      movel([0.344723, -1.349574, -2.579464, -0.783351, 1.570796, 1.915519],accel_mss,speed_ms,0,blend_radius_m)
      speed_ms = 0.003
      movel([0.344723, -1.359446, -2.584078, -0.768865, 1.570796, 1.915519],accel_mss,speed_ms,0,blend_radius_m)
      speed_ms = 0.007
      movel([0.344029, -1.359514, -2.584032, -0.768843, 1.570796, 1.914825],accel_mss,speed_ms,0,blend_radius_m)
      movel([0.343242, -1.359584, -2.583985, -0.768820, 1.570796, 1.914038],accel_mss,speed_ms,0,blend_radius_m)
      movel([0.342310, -1.359660, -2.583934, -0.768796, 1.570796, 1.913106],accel_mss,speed_ms,0,blend_radius_m)
      movel([0.339886, -1.359848, -2.583806, -0.768735, 1.570796, 1.910682],accel_mss,speed_ms,0,blend_radius_m)
      movel([0.340151, -1.359124, -2.584296, -0.768969, 1.570796, 1.910947],accel_mss,speed_ms,0,blend_radius_m)
      movel([0.340416, -1.358401, -2.584784, -0.769203, 1.570796, 1.911212],accel_mss,speed_ms,0,blend_radius_m)
      movel([0.342598, -1.358879, -2.584462, -0.769048, 1.570796, 1.913394],accel_mss,speed_ms,0,blend_radius_m)
      movel([0.343434, -1.359066, -2.584335, -0.768988, 1.570796, 1.914230],accel_mss,speed_ms,0,blend_radius_m)
      movel([0.344132, -1.359235, -2.584221, -0.768933, 1.570796, 1.914929],accel_mss,speed_ms,0,blend_radius_m)
      movel([0.344743, -1.359392, -2.584115, -0.768882, 1.570796, 1.915539],accel_mss,speed_ms,0,blend_radius_m)
      movel([0.344756, -1.359400, -2.584109, -0.768880, 1.570796, 1.915553],accel_mss,speed_ms,0,blend_radius_m)
      movel([0.344754, -1.359419, -2.584097, -0.768874, 1.570796, 1.915551],accel_mss,speed_ms,0,blend_radius_m)
      movel([0.344743, -1.359435, -2.584085, -0.768868, 1.570796, 1.915540],accel_mss,speed_ms,0,blend_radius_m)
      movel([0.344723, -1.359446, -2.584078, -0.768865, 1.570796, 1.915519],accel_mss,speed_ms,0,blend_radius_m)
      speed_ms = 0.003
      movel([0.344723, -1.362784, -2.585600, -0.764005, 1.570796, 1.915519],accel_mss,speed_ms,0,blend_radius_m)
      speed_ms = 0.007
      movel([0.344029, -1.362852, -2.585554, -0.763984, 1.570796, 1.914825],accel_mss,speed_ms,0,blend_radius_m)
      movel([0.343242, -1.362922, -2.585506, -0.763961, 1.570796, 1.914038],accel_mss,speed_ms,0,blend_radius_m)
      movel([0.342310, -1.362997, -2.585455, -0.763937, 1.570796, 1.913106],accel_mss,speed_ms,0,blend_radius_m)
      movel([0.339886, -1.363185, -2.585327, -0.763877, 1.570796, 1.910682],accel_mss,speed_ms,0,blend_radius_m)
      movel([0.340151, -1.362463, -2.585818, -0.764108, 1.570796, 1.910947],accel_mss,speed_ms,0,blend_radius_m)
      movel([0.340416, -1.361742, -2.586307, -0.764340, 1.570796, 1.911212],accel_mss,speed_ms,0,blend_radius_m)
      movel([0.342598, -1.362219, -2.585984, -0.764186, 1.570796, 1.913394],accel_mss,speed_ms,0,blend_radius_m)
      movel([0.343434, -1.362405, -2.585857, -0.764127, 1.570796, 1.914230],accel_mss,speed_ms,0,blend_radius_m)
      movel([0.344132, -1.362573, -2.585743, -0.764073, 1.570796, 1.914929],accel_mss,speed_ms,0,blend_radius_m)
      movel([0.344743, -1.362730, -2.585636, -0.764022, 1.570796, 1.915539],accel_mss,speed_ms,0,blend_radius_m)
      movel([0.344756, -1.362738, -2.585631, -0.764020, 1.570796, 1.915553],accel_mss,speed_ms,0,blend_radius_m)
      movel([0.344754, -1.362757, -2.585618, -0.764014, 1.570796, 1.915551],accel_mss,speed_ms,0,blend_radius_m)
      movel([0.344743, -1.362773, -2.585607, -0.764009, 1.570796, 1.915540],accel_mss,speed_ms,0,blend_radius_m)
      movel([0.344723, -1.362784, -2.585600, -0.764005, 1.570796, 1.915519],accel_mss,speed_ms,0,blend_radius_m)
      speed_ms = 0.003
      movel([0.344723, -1.349574, -2.579464, -0.783351, 1.570796, 1.915519],accel_mss,speed_ms,0,blend_radius_m)
      speed_ms = 0.01
      movel([0.344723, -1.324283, -2.566799, -0.821307, 1.570796, 1.915519],accel_mss,speed_ms,0,blend_radius_m)
      movel([0.344980, -1.321488, -2.568590, -0.822311, 1.570796, 1.915776],accel_mss,speed_ms,0,blend_radius_m)
      movel([0.344980, -1.346826, -2.581290, -0.784273, 1.570796, 1.915776],accel_mss,speed_ms,0,blend_radius_m)
      speed_ms = 0.003
      movel([0.344980, -1.356718, -2.585918, -0.769752, 1.570796, 1.915776],accel_mss,speed_ms,0,blend_radius_m)
      speed_ms = 0.007
      movel([0.344880, -1.356721, -2.585916, -0.769751, 1.570796, 1.915676],accel_mss,speed_ms,0,blend_radius_m)
      movel([0.344783, -1.356715, -2.585921, -0.769754, 1.570796, 1.915579],accel_mss,speed_ms,0,blend_radius_m)
      movel([0.344690, -1.356699, -2.585931, -0.769759, 1.570796, 1.915486],accel_mss,speed_ms,0,blend_radius_m)
      movel([0.320621, -1.351621, -2.589329, -0.771439, 1.570796, 1.891418],accel_mss,speed_ms,0,blend_radius_m)
      movel([0.295950, -1.347201, -2.592258, -0.772930, 1.570796, 1.866746],accel_mss,speed_ms,0,blend_radius_m)
      movel([0.295898, -1.347189, -2.592266, -0.772934, 1.570796, 1.866695],accel_mss,speed_ms,0,blend_radius_m)
      movel([0.295858, -1.347164, -2.592282, -0.772943, 1.570796, 1.866654],accel_mss,speed_ms,0,blend_radius_m)
      movel([0.295822, -1.347135, -2.592301, -0.772953, 1.570796, 1.866618],accel_mss,speed_ms,0,blend_radius_m)
      movel([0.295809, -1.347107, -2.592320, -0.772962, 1.570796, 1.866606],accel_mss,speed_ms,0,blend_radius_m)
      movel([0.295812, -1.347070, -2.592344, -0.772975, 1.570796, 1.866608],accel_mss,speed_ms,0,blend_radius_m)
      movel([0.295826, -1.347031, -2.592369, -0.772988, 1.570796, 1.866623],accel_mss,speed_ms,0,blend_radius_m)
      movel([0.300073, -1.339721, -2.597152, -0.775516, 1.570796, 1.870870],accel_mss,speed_ms,0,blend_radius_m)
      movel([0.304360, -1.332369, -2.601889, -0.778132, 1.570796, 1.875156],accel_mss,speed_ms,0,blend_radius_m)
      movel([0.304408, -1.332297, -2.601935, -0.778157, 1.570796, 1.875204],accel_mss,speed_ms,0,blend_radius_m)
      movel([0.304466, -1.332229, -2.601978, -0.778182, 1.570796, 1.875263],accel_mss,speed_ms,0,blend_radius_m)
      movel([0.304533, -1.332167, -2.602018, -0.778204, 1.570796, 1.875329],accel_mss,speed_ms,0,blend_radius_m)
      movel([0.304566, -1.332146, -2.602031, -0.778212, 1.570796, 1.875363],accel_mss,speed_ms,0,blend_radius_m)
      movel([0.304602, -1.332142, -2.602034, -0.778213, 1.570796, 1.875398],accel_mss,speed_ms,0,blend_radius_m)
      movel([0.306078, -1.332291, -2.601938, -0.778159, 1.570796, 1.876875],accel_mss,speed_ms,0,blend_radius_m)
      movel([0.307729, -1.332470, -2.601824, -0.778095, 1.570796, 1.878525],accel_mss,speed_ms,0,blend_radius_m)
      movel([0.309667, -1.332702, -2.601676, -0.778011, 1.570796, 1.880463],accel_mss,speed_ms,0,blend_radius_m)
      movel([0.315690, -1.333471, -2.601183, -0.777735, 1.570796, 1.886487],accel_mss,speed_ms,0,blend_radius_m)
      movel([0.321678, -1.334295, -2.600655, -0.777439, 1.570796, 1.892474],accel_mss,speed_ms,0,blend_radius_m)
      movel([0.323791, -1.334609, -2.600453, -0.777327, 1.570796, 1.894587],accel_mss,speed_ms,0,blend_radius_m)
      movel([0.325891, -1.334945, -2.600237, -0.777207, 1.570796, 1.896687],accel_mss,speed_ms,0,blend_radius_m)
      movel([0.327973, -1.335306, -2.600005, -0.777078, 1.570796, 1.898769],accel_mss,speed_ms,0,blend_radius_m)
      movel([0.329039, -1.335506, -2.599877, -0.777006, 1.570796, 1.899836],accel_mss,speed_ms,0,blend_radius_m)
      movel([0.330096, -1.335717, -2.599741, -0.776931, 1.570796, 1.900893],accel_mss,speed_ms,0,blend_radius_m)
      movel([0.331144, -1.335944, -2.599595, -0.776850, 1.570796, 1.901941],accel_mss,speed_ms,0,blend_radius_m)
      movel([0.332182, -1.336185, -2.599439, -0.776764, 1.570796, 1.902978],accel_mss,speed_ms,0,blend_radius_m)
      movel([0.333127, -1.336420, -2.599288, -0.776681, 1.570796, 1.903923],accel_mss,speed_ms,0,blend_radius_m)
      movel([0.334059, -1.336671, -2.599126, -0.776592, 1.570796, 1.904855],accel_mss,speed_ms,0,blend_radius_m)
      movel([0.334978, -1.336941, -2.598952, -0.776496, 1.570796, 1.905774],accel_mss,speed_ms,0,blend_radius_m)
      movel([0.335887, -1.337224, -2.598769, -0.776396, 1.570796, 1.906684],accel_mss,speed_ms,0,blend_radius_m)
      movel([0.336686, -1.337490, -2.598597, -0.776302, 1.570796, 1.907483],accel_mss,speed_ms,0,blend_radius_m)
      movel([0.337471, -1.337775, -2.598413, -0.776201, 1.570796, 1.908267],accel_mss,speed_ms,0,blend_radius_m)
      movel([0.338245, -1.338072, -2.598221, -0.776096, 1.570796, 1.909041],accel_mss,speed_ms,0,blend_radius_m)
      movel([0.339005, -1.338388, -2.598016, -0.775984, 1.570796, 1.909801],accel_mss,speed_ms,0,blend_radius_m)
      movel([0.339755, -1.338718, -2.597803, -0.775868, 1.570796, 1.910551],accel_mss,speed_ms,0,blend_radius_m)
      movel([0.340490, -1.339065, -2.597578, -0.775746, 1.570796, 1.911286],accel_mss,speed_ms,0,blend_radius_m)
      movel([0.341213, -1.339426, -2.597344, -0.775619, 1.570796, 1.912009],accel_mss,speed_ms,0,blend_radius_m)
      movel([0.341919, -1.339803, -2.597099, -0.775487, 1.570796, 1.912715],accel_mss,speed_ms,0,blend_radius_m)
      movel([0.342412, -1.340083, -2.596917, -0.775389, 1.570796, 1.913209],accel_mss,speed_ms,0,blend_radius_m)
      movel([0.342888, -1.340385, -2.596721, -0.775283, 1.570796, 1.913685],accel_mss,speed_ms,0,blend_radius_m)
      movel([0.343349, -1.340701, -2.596515, -0.775173, 1.570796, 1.914145],accel_mss,speed_ms,0,blend_radius_m)
      movel([0.343790, -1.341036, -2.596297, -0.775056, 1.570796, 1.914586],accel_mss,speed_ms,0,blend_radius_m)
      movel([0.344215, -1.341389, -2.596067, -0.774933, 1.570796, 1.915011],accel_mss,speed_ms,0,blend_radius_m)
      movel([0.344625, -1.341755, -2.595829, -0.774805, 1.570796, 1.915421],accel_mss,speed_ms,0,blend_radius_m)
      movel([0.345013, -1.342139, -2.595579, -0.774672, 1.570796, 1.915809],accel_mss,speed_ms,0,blend_radius_m)
      movel([0.345385, -1.342540, -2.595316, -0.774532, 1.570796, 1.916181],accel_mss,speed_ms,0,blend_radius_m)
      movel([0.345737, -1.342955, -2.595045, -0.774388, 1.570796, 1.916534],accel_mss,speed_ms,0,blend_radius_m)
      movel([0.345992, -1.343283, -2.594831, -0.774275, 1.570796, 1.916789],accel_mss,speed_ms,0,blend_radius_m)
      movel([0.346229, -1.343625, -2.594607, -0.774157, 1.570796, 1.917026],accel_mss,speed_ms,0,blend_radius_m)
      movel([0.346450, -1.343978, -2.594376, -0.774035, 1.570796, 1.917247],accel_mss,speed_ms,0,blend_radius_m)
      movel([0.346655, -1.344344, -2.594136, -0.773909, 1.570796, 1.917451],accel_mss,speed_ms,0,blend_radius_m)
      movel([0.346843, -1.344721, -2.593889, -0.773779, 1.570796, 1.917639],accel_mss,speed_ms,0,blend_radius_m)
      movel([0.347014, -1.345108, -2.593635, -0.773646, 1.570796, 1.917811],accel_mss,speed_ms,0,blend_radius_m)
      movel([0.347168, -1.345505, -2.593374, -0.773510, 1.570796, 1.917964],accel_mss,speed_ms,0,blend_radius_m)
      movel([0.347305, -1.345913, -2.593106, -0.773370, 1.570796, 1.918102],accel_mss,speed_ms,0,blend_radius_m)
      movel([0.347424, -1.346332, -2.592830, -0.773227, 1.570796, 1.918221],accel_mss,speed_ms,0,blend_radius_m)
      movel([0.347525, -1.346761, -2.592548, -0.773080, 1.570796, 1.918321],accel_mss,speed_ms,0,blend_radius_m)
      movel([0.347605, -1.347180, -2.592272, -0.772938, 1.570796, 1.918401],accel_mss,speed_ms,0,blend_radius_m)
      movel([0.347668, -1.347607, -2.591990, -0.772792, 1.570796, 1.918464],accel_mss,speed_ms,0,blend_radius_m)
      movel([0.347707, -1.348044, -2.591701, -0.772644, 1.570796, 1.918504],accel_mss,speed_ms,0,blend_radius_m)
      movel([0.347731, -1.348488, -2.591408, -0.772493, 1.570796, 1.918527],accel_mss,speed_ms,0,blend_radius_m)
      movel([0.347733, -1.348942, -2.591108, -0.772340, 1.570796, 1.918529],accel_mss,speed_ms,0,blend_radius_m)
      movel([0.347720, -1.349399, -2.590805, -0.772185, 1.570796, 1.918516],accel_mss,speed_ms,0,blend_radius_m)
      movel([0.347684, -1.349864, -2.590496, -0.772028, 1.570796, 1.918481],accel_mss,speed_ms,0,blend_radius_m)
      movel([0.347630, -1.350336, -2.590184, -0.771870, 1.570796, 1.918426],accel_mss,speed_ms,0,blend_radius_m)
      movel([0.347558, -1.350810, -2.589868, -0.771710, 1.570796, 1.918354],accel_mss,speed_ms,0,blend_radius_m)
      movel([0.347467, -1.351290, -2.589549, -0.771549, 1.570796, 1.918263],accel_mss,speed_ms,0,blend_radius_m)
      movel([0.347400, -1.351565, -2.589366, -0.771457, 1.570796, 1.918196],accel_mss,speed_ms,0,blend_radius_m)
      movel([0.347318, -1.351842, -2.589182, -0.771365, 1.570796, 1.918115],accel_mss,speed_ms,0,blend_radius_m)
      movel([0.347219, -1.352121, -2.588996, -0.771272, 1.570796, 1.918015],accel_mss,speed_ms,0,blend_radius_m)
      movel([0.346861, -1.353037, -2.588385, -0.770967, 1.570796, 1.917658],accel_mss,speed_ms,0,blend_radius_m)
      movel([0.346494, -1.353953, -2.587773, -0.770663, 1.570796, 1.917291],accel_mss,speed_ms,0,blend_radius_m)
      movel([0.346110, -1.354891, -2.587145, -0.770353, 1.570796, 1.916906],accel_mss,speed_ms,0,blend_radius_m)
      movel([0.345719, -1.355829, -2.586516, -0.770044, 1.570796, 1.916515],accel_mss,speed_ms,0,blend_radius_m)
      movel([0.345654, -1.355967, -2.586424, -0.769999, 1.570796, 1.916450],accel_mss,speed_ms,0,blend_radius_m)
      movel([0.345581, -1.356105, -2.586331, -0.769953, 1.570796, 1.916377],accel_mss,speed_ms,0,blend_radius_m)
      movel([0.345495, -1.356240, -2.586240, -0.769909, 1.570796, 1.916292],accel_mss,speed_ms,0,blend_radius_m)
      movel([0.345403, -1.356375, -2.586149, -0.769865, 1.570796, 1.916199],accel_mss,speed_ms,0,blend_radius_m)
      movel([0.345351, -1.356438, -2.586107, -0.769844, 1.570796, 1.916147],accel_mss,speed_ms,0,blend_radius_m)
      movel([0.345294, -1.356502, -2.586064, -0.769823, 1.570796, 1.916090],accel_mss,speed_ms,0,blend_radius_m)
      movel([0.345238, -1.356559, -2.586025, -0.769804, 1.570796, 1.916034],accel_mss,speed_ms,0,blend_radius_m)
      movel([0.345175, -1.356612, -2.585990, -0.769787, 1.570796, 1.915972],accel_mss,speed_ms,0,blend_radius_m)
      movel([0.345123, -1.356652, -2.585963, -0.769774, 1.570796, 1.915919],accel_mss,speed_ms,0,blend_radius_m)
      movel([0.345067, -1.356689, -2.585938, -0.769762, 1.570796, 1.915863],accel_mss,speed_ms,0,blend_radius_m)
      movel([0.345023, -1.356710, -2.585924, -0.769755, 1.570796, 1.915820],accel_mss,speed_ms,0,blend_radius_m)
      movel([0.344980, -1.356718, -2.585918, -0.769752, 1.570796, 1.915776],accel_mss,speed_ms,0,blend_radius_m)
      speed_ms = 0.003
      movel([0.344980, -1.360063, -2.587444, -0.764881, 1.570796, 1.915776],accel_mss,speed_ms,0,blend_radius_m)
      speed_ms = 0.007
      movel([0.344880, -1.360066, -2.587442, -0.764880, 1.570796, 1.915676],accel_mss,speed_ms,0,blend_radius_m)
      movel([0.344783, -1.360060, -2.587447, -0.764882, 1.570796, 1.915579],accel_mss,speed_ms,0,blend_radius_m)
      movel([0.344690, -1.360044, -2.587457, -0.764888, 1.570796, 1.915486],accel_mss,speed_ms,0,blend_radius_m)
      movel([0.320621, -1.354979, -2.590864, -0.766546, 1.570796, 1.891418],accel_mss,speed_ms,0,blend_radius_m)
      movel([0.295950, -1.350570, -2.593800, -0.768019, 1.570796, 1.866746],accel_mss,speed_ms,0,blend_radius_m)
      movel([0.295898, -1.350559, -2.593807, -0.768023, 1.570796, 1.866695],accel_mss,speed_ms,0,blend_radius_m)
      movel([0.295858, -1.350534, -2.593824, -0.768031, 1.570796, 1.866654],accel_mss,speed_ms,0,blend_radius_m)
      movel([0.295822, -1.350504, -2.593843, -0.768041, 1.570796, 1.866618],accel_mss,speed_ms,0,blend_radius_m)
      movel([0.295809, -1.350476, -2.593862, -0.768051, 1.570796, 1.866606],accel_mss,speed_ms,0,blend_radius_m)
      movel([0.295812, -1.350440, -2.593886, -0.768063, 1.570796, 1.866608],accel_mss,speed_ms,0,blend_radius_m)
      movel([0.295826, -1.350401, -2.593912, -0.768076, 1.570796, 1.866623],accel_mss,speed_ms,0,blend_radius_m)
      movel([0.300073, -1.343109, -2.598706, -0.770573, 1.570796, 1.870870],accel_mss,speed_ms,0,blend_radius_m)
      movel([0.304360, -1.335775, -2.603456, -0.773158, 1.570796, 1.875156],accel_mss,speed_ms,0,blend_radius_m)
      movel([0.304408, -1.335704, -2.603501, -0.773184, 1.570796, 1.875204],accel_mss,speed_ms,0,blend_radius_m)
      movel([0.304466, -1.335636, -2.603545, -0.773208, 1.570796, 1.875263],accel_mss,speed_ms,0,blend_radius_m)
      movel([0.304533, -1.335574, -2.603585, -0.773230, 1.570796, 1.875329],accel_mss,speed_ms,0,blend_radius_m)
      movel([0.304566, -1.335553, -2.603598, -0.773238, 1.570796, 1.875363],accel_mss,speed_ms,0,blend_radius_m)
      movel([0.304602, -1.335549, -2.603601, -0.773239, 1.570796, 1.875398],accel_mss,speed_ms,0,blend_radius_m)
      movel([0.306078, -1.335698, -2.603505, -0.773186, 1.570796, 1.876875],accel_mss,speed_ms,0,blend_radius_m)
      movel([0.307729, -1.335876, -2.603390, -0.773122, 1.570796, 1.878525],accel_mss,speed_ms,0,blend_radius_m)
      movel([0.309667, -1.336108, -2.603242, -0.773040, 1.570796, 1.880463],accel_mss,speed_ms,0,blend_radius_m)
      movel([0.315690, -1.336875, -2.602748, -0.772766, 1.570796, 1.886487],accel_mss,speed_ms,0,blend_radius_m)
      movel([0.321678, -1.337697, -2.602218, -0.772474, 1.570796, 1.892474],accel_mss,speed_ms,0,blend_radius_m)
      movel([0.323791, -1.338010, -2.602016, -0.772363, 1.570796, 1.894587],accel_mss,speed_ms,0,blend_radius_m)
      movel([0.325891, -1.338345, -2.601800, -0.772244, 1.570796, 1.896687],accel_mss,speed_ms,0,blend_radius_m)
      movel([0.327973, -1.338705, -2.601567, -0.772117, 1.570796, 1.898769],accel_mss,speed_ms,0,blend_radius_m)
      movel([0.329039, -1.338904, -2.601438, -0.772046, 1.570796, 1.899836],accel_mss,speed_ms,0,blend_radius_m)
      movel([0.330096, -1.339115, -2.601302, -0.771972, 1.570796, 1.900893],accel_mss,speed_ms,0,blend_radius_m)
      movel([0.331144, -1.339342, -2.601155, -0.771892, 1.570796, 1.901941],accel_mss,speed_ms,0,blend_radius_m)
      movel([0.332182, -1.339582, -2.600999, -0.771807, 1.570796, 1.902978],accel_mss,speed_ms,0,blend_radius_m)
      movel([0.333127, -1.339817, -2.600848, -0.771725, 1.570796, 1.903923],accel_mss,speed_ms,0,blend_radius_m)
      movel([0.334059, -1.340067, -2.600685, -0.771637, 1.570796, 1.904855],accel_mss,speed_ms,0,blend_radius_m)
      movel([0.334978, -1.340336, -2.600511, -0.771542, 1.570796, 1.905774],accel_mss,speed_ms,0,blend_radius_m)
      movel([0.335887, -1.340619, -2.600328, -0.771443, 1.570796, 1.906684],accel_mss,speed_ms,0,blend_radius_m)
      movel([0.336686, -1.340884, -2.600155, -0.771350, 1.570796, 1.907483],accel_mss,speed_ms,0,blend_radius_m)
      movel([0.337471, -1.341168, -2.599971, -0.771250, 1.570796, 1.908267],accel_mss,speed_ms,0,blend_radius_m)
      movel([0.338245, -1.341465, -2.599778, -0.771146, 1.570796, 1.909041],accel_mss,speed_ms,0,blend_radius_m)
      movel([0.339005, -1.341780, -2.599573, -0.771036, 1.570796, 1.909801],accel_mss,speed_ms,0,blend_radius_m)
      movel([0.339755, -1.342108, -2.599359, -0.770922, 1.570796, 1.910551],accel_mss,speed_ms,0,blend_radius_m)
      movel([0.340490, -1.342455, -2.599133, -0.770801, 1.570796, 1.911286],accel_mss,speed_ms,0,blend_radius_m)
      movel([0.341213, -1.342815, -2.598899, -0.770676, 1.570796, 1.912009],accel_mss,speed_ms,0,blend_radius_m)
      movel([0.341919, -1.343191, -2.598653, -0.770545, 1.570796, 1.912715],accel_mss,speed_ms,0,blend_radius_m)
      movel([0.342412, -1.343471, -2.598471, -0.770448, 1.570796, 1.913209],accel_mss,speed_ms,0,blend_radius_m)
      movel([0.342888, -1.343771, -2.598274, -0.770343, 1.570796, 1.913685],accel_mss,speed_ms,0,blend_radius_m)
      movel([0.343349, -1.344087, -2.598068, -0.770234, 1.570796, 1.914145],accel_mss,speed_ms,0,blend_radius_m)
      movel([0.343790, -1.344421, -2.597849, -0.770118, 1.570796, 1.914586],accel_mss,speed_ms,0,blend_radius_m)
      movel([0.344215, -1.344773, -2.597619, -0.769997, 1.570796, 1.915011],accel_mss,speed_ms,0,blend_radius_m)
      movel([0.344625, -1.345138, -2.597380, -0.769871, 1.570796, 1.915421],accel_mss,speed_ms,0,blend_radius_m)
      movel([0.345013, -1.345521, -2.597129, -0.769739, 1.570796, 1.915809],accel_mss,speed_ms,0,blend_radius_m)
      movel([0.345385, -1.345922, -2.596866, -0.769601, 1.570796, 1.916181],accel_mss,speed_ms,0,blend_radius_m)
      movel([0.345737, -1.346336, -2.596594, -0.769459, 1.570796, 1.916534],accel_mss,speed_ms,0,blend_radius_m)
      movel([0.345992, -1.346662, -2.596380, -0.769347, 1.570796, 1.916789],accel_mss,speed_ms,0,blend_radius_m)
      movel([0.346229, -1.347004, -2.596155, -0.769230, 1.570796, 1.917026],accel_mss,speed_ms,0,blend_radius_m)
      movel([0.346450, -1.347356, -2.595923, -0.769110, 1.570796, 1.917247],accel_mss,speed_ms,0,blend_radius_m)
      movel([0.346655, -1.347721, -2.595683, -0.768985, 1.570796, 1.917451],accel_mss,speed_ms,0,blend_radius_m)
      movel([0.346843, -1.348097, -2.595435, -0.768857, 1.570796, 1.917639],accel_mss,speed_ms,0,blend_radius_m)
      movel([0.347014, -1.348483, -2.595180, -0.768726, 1.570796, 1.917811],accel_mss,speed_ms,0,blend_radius_m)
      movel([0.347168, -1.348879, -2.594919, -0.768591, 1.570796, 1.917964],accel_mss,speed_ms,0,blend_radius_m)
      movel([0.347305, -1.349286, -2.594650, -0.768453, 1.570796, 1.918102],accel_mss,speed_ms,0,blend_radius_m)
      movel([0.347424, -1.349704, -2.594374, -0.768312, 1.570796, 1.918221],accel_mss,speed_ms,0,blend_radius_m)
      movel([0.347525, -1.350132, -2.594090, -0.768167, 1.570796, 1.918321],accel_mss,speed_ms,0,blend_radius_m)
      movel([0.347605, -1.350549, -2.593813, -0.768026, 1.570796, 1.918401],accel_mss,speed_ms,0,blend_radius_m)
      movel([0.347668, -1.350975, -2.593531, -0.767883, 1.570796, 1.918464],accel_mss,speed_ms,0,blend_radius_m)
      movel([0.347707, -1.351412, -2.593241, -0.767736, 1.570796, 1.918504],accel_mss,speed_ms,0,blend_radius_m)
      movel([0.347731, -1.351854, -2.592948, -0.767587, 1.570796, 1.918527],accel_mss,speed_ms,0,blend_radius_m)
      movel([0.347733, -1.352307, -2.592646, -0.767436, 1.570796, 1.918529],accel_mss,speed_ms,0,blend_radius_m)
      movel([0.347720, -1.352763, -2.592343, -0.767283, 1.570796, 1.918516],accel_mss,speed_ms,0,blend_radius_m)
      movel([0.347684, -1.353227, -2.592034, -0.767128, 1.570796, 1.918481],accel_mss,speed_ms,0,blend_radius_m)
      movel([0.347630, -1.353697, -2.591720, -0.766972, 1.570796, 1.918426],accel_mss,speed_ms,0,blend_radius_m)
      movel([0.347558, -1.354170, -2.591404, -0.766814, 1.570796, 1.918354],accel_mss,speed_ms,0,blend_radius_m)
      movel([0.347467, -1.354649, -2.591084, -0.766655, 1.570796, 1.918263],accel_mss,speed_ms,0,blend_radius_m)
      movel([0.347400, -1.354924, -2.590901, -0.766564, 1.570796, 1.918196],accel_mss,speed_ms,0,blend_radius_m)
      movel([0.347318, -1.355199, -2.590716, -0.766473, 1.570796, 1.918115],accel_mss,speed_ms,0,blend_radius_m)
      movel([0.347219, -1.355478, -2.590530, -0.766381, 1.570796, 1.918015],accel_mss,speed_ms,0,blend_radius_m)
      movel([0.346861, -1.356392, -2.589917, -0.766080, 1.570796, 1.917658],accel_mss,speed_ms,0,blend_radius_m)
      movel([0.346494, -1.357305, -2.589304, -0.765780, 1.570796, 1.917291],accel_mss,speed_ms,0,blend_radius_m)
      movel([0.346110, -1.358241, -2.588674, -0.765474, 1.570796, 1.916906],accel_mss,speed_ms,0,blend_radius_m)
      movel([0.345719, -1.359176, -2.588044, -0.765169, 1.570796, 1.916515],accel_mss,speed_ms,0,blend_radius_m)
      movel([0.345654, -1.359314, -2.587951, -0.765124, 1.570796, 1.916450],accel_mss,speed_ms,0,blend_radius_m)
      movel([0.345581, -1.359452, -2.587858, -0.765080, 1.570796, 1.916377],accel_mss,speed_ms,0,blend_radius_m)
      movel([0.345495, -1.359586, -2.587767, -0.765036, 1.570796, 1.916292],accel_mss,speed_ms,0,blend_radius_m)
      movel([0.345403, -1.359721, -2.587676, -0.764992, 1.570796, 1.916199],accel_mss,speed_ms,0,blend_radius_m)
      movel([0.345351, -1.359784, -2.587633, -0.764972, 1.570796, 1.916147],accel_mss,speed_ms,0,blend_radius_m)
      movel([0.345294, -1.359848, -2.587590, -0.764951, 1.570796, 1.916090],accel_mss,speed_ms,0,blend_radius_m)
      movel([0.345238, -1.359905, -2.587552, -0.764933, 1.570796, 1.916034],accel_mss,speed_ms,0,blend_radius_m)
      movel([0.345175, -1.359957, -2.587516, -0.764916, 1.570796, 1.915972],accel_mss,speed_ms,0,blend_radius_m)
      movel([0.345123, -1.359998, -2.587489, -0.764903, 1.570796, 1.915919],accel_mss,speed_ms,0,blend_radius_m)
      movel([0.345067, -1.360034, -2.587464, -0.764891, 1.570796, 1.915863],accel_mss,speed_ms,0,blend_radius_m)
      movel([0.345023, -1.360055, -2.587450, -0.764884, 1.570796, 1.915820],accel_mss,speed_ms,0,blend_radius_m)
      movel([0.344980, -1.360063, -2.587444, -0.764881, 1.570796, 1.915776],accel_mss,speed_ms,0,blend_radius_m)
      speed_ms = 0.003
      movel([0.344980, -1.346826, -2.581290, -0.784273, 1.570796, 1.915776],accel_mss,speed_ms,0,blend_radius_m)
      speed_ms = 0.01
      movel([0.344980, -1.321488, -2.568590, -0.822311, 1.570796, 1.915776],accel_mss,speed_ms,0,blend_radius_m)
      movel([0.342353, -1.326735, -2.565220, -0.820435, 1.570796, 1.913150],accel_mss,speed_ms,0,blend_radius_m)
      movel([0.342353, -1.351985, -2.577853, -0.782552, 1.570796, 1.913150],accel_mss,speed_ms,0,blend_radius_m)
      speed_ms = 0.003
      movel([0.342353, -1.361839, -2.582456, -0.768095, 1.570796, 1.913150],accel_mss,speed_ms,0,blend_radius_m)
      speed_ms = 0.007
      movel([0.341641, -1.363771, -2.581139, -0.767479, 1.570796, 1.912437],accel_mss,speed_ms,0,blend_radius_m)
      movel([0.340931, -1.365698, -2.579822, -0.766870, 1.570796, 1.911728],accel_mss,speed_ms,0,blend_radius_m)
      movel([0.336123, -1.366174, -2.579495, -0.766720, 1.570796, 1.906919],accel_mss,speed_ms,0,blend_radius_m)
      movel([0.334430, -1.366357, -2.579369, -0.766663, 1.570796, 1.905226],accel_mss,speed_ms,0,blend_radius_m)
      movel([0.332727, -1.366563, -2.579228, -0.766598, 1.570796, 1.903523],accel_mss,speed_ms,0,blend_radius_m)
      movel([0.331393, -1.366752, -2.579098, -0.766539, 1.570796, 1.902189],accel_mss,speed_ms,0,blend_radius_m)
      movel([0.330047, -1.366975, -2.578945, -0.766469, 1.570796, 1.900843],accel_mss,speed_ms,0,blend_radius_m)
      movel([0.328764, -1.367221, -2.578776, -0.766392, 1.570796, 1.899560],accel_mss,speed_ms,0,blend_radius_m)
      movel([0.327473, -1.367502, -2.578582, -0.766304, 1.570796, 1.898270],accel_mss,speed_ms,0,blend_radius_m)
      movel([0.325956, -1.367865, -2.578333, -0.766191, 1.570796, 1.896752],accel_mss,speed_ms,0,blend_radius_m)
      movel([0.324433, -1.368257, -2.578063, -0.766069, 1.570796, 1.895230],accel_mss,speed_ms,0,blend_radius_m)
      movel([0.323162, -1.368604, -2.577824, -0.765961, 1.570796, 1.893958],accel_mss,speed_ms,0,blend_radius_m)
      movel([0.321888, -1.368978, -2.577566, -0.765845, 1.570796, 1.892684],accel_mss,speed_ms,0,blend_radius_m)
      movel([0.320612, -1.369374, -2.577293, -0.765722, 1.570796, 1.891408],accel_mss,speed_ms,0,blend_radius_m)
      movel([0.319335, -1.369795, -2.577002, -0.765592, 1.570796, 1.890132],accel_mss,speed_ms,0,blend_radius_m)
      movel([0.318059, -1.370240, -2.576694, -0.765455, 1.570796, 1.888855],accel_mss,speed_ms,0,blend_radius_m)
      movel([0.316792, -1.370704, -2.576373, -0.765312, 1.570796, 1.887588],accel_mss,speed_ms,0,blend_radius_m)
      movel([0.315526, -1.371191, -2.576035, -0.765162, 1.570796, 1.886322],accel_mss,speed_ms,0,blend_radius_m)
      movel([0.314261, -1.371704, -2.575680, -0.765005, 1.570796, 1.885058],accel_mss,speed_ms,0,blend_radius_m)
      movel([0.312998, -1.372237, -2.575310, -0.764842, 1.570796, 1.883794],accel_mss,speed_ms,0,blend_radius_m)
      movel([0.311739, -1.372792, -2.574924, -0.764673, 1.570796, 1.882536],accel_mss,speed_ms,0,blend_radius_m)
      movel([0.310506, -1.373361, -2.574529, -0.764500, 1.570796, 1.881302],accel_mss,speed_ms,0,blend_radius_m)
      movel([0.309278, -1.373949, -2.574119, -0.764321, 1.570796, 1.880074],accel_mss,speed_ms,0,blend_radius_m)
      movel([0.308056, -1.374560, -2.573693, -0.764136, 1.570796, 1.878852],accel_mss,speed_ms,0,blend_radius_m)
      movel([0.306839, -1.375192, -2.573251, -0.763945, 1.570796, 1.877635],accel_mss,speed_ms,0,blend_radius_m)
      movel([0.305626, -1.375845, -2.572795, -0.763749, 1.570796, 1.876423],accel_mss,speed_ms,0,blend_radius_m)
      movel([0.304459, -1.376497, -2.572338, -0.763554, 1.570796, 1.875255],accel_mss,speed_ms,0,blend_radius_m)
      movel([0.303297, -1.377173, -2.571865, -0.763352, 1.570796, 1.874093],accel_mss,speed_ms,0,blend_radius_m)
      movel([0.302144, -1.377865, -2.571378, -0.763145, 1.570796, 1.872941],accel_mss,speed_ms,0,blend_radius_m)
      movel([0.301002, -1.378581, -2.570875, -0.762933, 1.570796, 1.871798],accel_mss,speed_ms,0,blend_radius_m)
      movel([0.299869, -1.379313, -2.570360, -0.762716, 1.570796, 1.870665],accel_mss,speed_ms,0,blend_radius_m)
      movel([0.299135, -1.379808, -2.570010, -0.762570, 1.570796, 1.869931],accel_mss,speed_ms,0,blend_radius_m)
      movel([0.298406, -1.380316, -2.569652, -0.762421, 1.570796, 1.869202],accel_mss,speed_ms,0,blend_radius_m)
      movel([0.297686, -1.380836, -2.569285, -0.762268, 1.570796, 1.868482],accel_mss,speed_ms,0,blend_radius_m)
      movel([0.296342, -1.381838, -2.568576, -0.761975, 1.570796, 1.867138],accel_mss,speed_ms,0,blend_radius_m)
      movel([0.295013, -1.382858, -2.567853, -0.761678, 1.570796, 1.865810],accel_mss,speed_ms,0,blend_radius_m)
      movel([0.293697, -1.383898, -2.567114, -0.761377, 1.570796, 1.864493],accel_mss,speed_ms,0,blend_radius_m)
      movel([0.292396, -1.384952, -2.566363, -0.761074, 1.570796, 1.863193],accel_mss,speed_ms,0,blend_radius_m)
      movel([0.291708, -1.385525, -2.565955, -0.760909, 1.570796, 1.862504],accel_mss,speed_ms,0,blend_radius_m)
      movel([0.291033, -1.386110, -2.565537, -0.760742, 1.570796, 1.861829],accel_mss,speed_ms,0,blend_radius_m)
      movel([0.290369, -1.386703, -2.565113, -0.760573, 1.570796, 1.861165],accel_mss,speed_ms,0,blend_radius_m)
      movel([0.289528, -1.387480, -2.564557, -0.760352, 1.570796, 1.860324],accel_mss,speed_ms,0,blend_radius_m)
      movel([0.288705, -1.388267, -2.563993, -0.760129, 1.570796, 1.859502],accel_mss,speed_ms,0,blend_radius_m)
      movel([0.287899, -1.389064, -2.563420, -0.759904, 1.570796, 1.858695],accel_mss,speed_ms,0,blend_radius_m)
      movel([0.287109, -1.389872, -2.562839, -0.759678, 1.570796, 1.857905],accel_mss,speed_ms,0,blend_radius_m)
      movel([0.286337, -1.390690, -2.562250, -0.759449, 1.570796, 1.857133],accel_mss,speed_ms,0,blend_radius_m)
      movel([0.285582, -1.391516, -2.561654, -0.759219, 1.570796, 1.856378],accel_mss,speed_ms,0,blend_radius_m)
      movel([0.284855, -1.392342, -2.561057, -0.758990, 1.570796, 1.855651],accel_mss,speed_ms,0,blend_radius_m)
      movel([0.284146, -1.393174, -2.560454, -0.758761, 1.570796, 1.854942],accel_mss,speed_ms,0,blend_radius_m)
      movel([0.283459, -1.394015, -2.559844, -0.758529, 1.570796, 1.854256],accel_mss,speed_ms,0,blend_radius_m)
      movel([0.282791, -1.394862, -2.559229, -0.758298, 1.570796, 1.853587],accel_mss,speed_ms,0,blend_radius_m)
      movel([0.282143, -1.395716, -2.558608, -0.758065, 1.570796, 1.852939],accel_mss,speed_ms,0,blend_radius_m)
      movel([0.281518, -1.396575, -2.557982, -0.757833, 1.570796, 1.852314],accel_mss,speed_ms,0,blend_radius_m)
      movel([0.280925, -1.397421, -2.557364, -0.757604, 1.570796, 1.851721],accel_mss,speed_ms,0,blend_radius_m)
      movel([0.280356, -1.398271, -2.556742, -0.757376, 1.570796, 1.851152],accel_mss,speed_ms,0,blend_radius_m)
      movel([0.279807, -1.399127, -2.556115, -0.757147, 1.570796, 1.850603],accel_mss,speed_ms,0,blend_radius_m)
      movel([0.279280, -1.399983, -2.555487, -0.756919, 1.570796, 1.850077],accel_mss,speed_ms,0,blend_radius_m)
      movel([0.278776, -1.400844, -2.554853, -0.756691, 1.570796, 1.849572],accel_mss,speed_ms,0,blend_radius_m)
      movel([0.278297, -1.401705, -2.554219, -0.756464, 1.570796, 1.849094],accel_mss,speed_ms,0,blend_radius_m)
      movel([0.277915, -1.402424, -2.553689, -0.756276, 1.570796, 1.848711],accel_mss,speed_ms,0,blend_radius_m)
      movel([0.277553, -1.403144, -2.553157, -0.756088, 1.570796, 1.848349],accel_mss,speed_ms,0,blend_radius_m)
      movel([0.277207, -1.403866, -2.552623, -0.755900, 1.570796, 1.848003],accel_mss,speed_ms,0,blend_radius_m)
      movel([0.276882, -1.404584, -2.552091, -0.755714, 1.570796, 1.847679],accel_mss,speed_ms,0,blend_radius_m)
      movel([0.276573, -1.405304, -2.551557, -0.755528, 1.570796, 1.847370],accel_mss,speed_ms,0,blend_radius_m)
      movel([0.276285, -1.406023, -2.551023, -0.755343, 1.570796, 1.847081],accel_mss,speed_ms,0,blend_radius_m)
      movel([0.276016, -1.406739, -2.550490, -0.755160, 1.570796, 1.846812],accel_mss,speed_ms,0,blend_radius_m)
      movel([0.275694, -1.407658, -2.549805, -0.754925, 1.570796, 1.846490],accel_mss,speed_ms,0,blend_radius_m)
      movel([0.275399, -1.408571, -2.549124, -0.754694, 1.570796, 1.846196],accel_mss,speed_ms,0,blend_radius_m)
      movel([0.275130, -1.409482, -2.548443, -0.754464, 1.570796, 1.845926],accel_mss,speed_ms,0,blend_radius_m)
      movel([0.274626, -1.411315, -2.547068, -0.754006, 1.570796, 1.845423],accel_mss,speed_ms,0,blend_radius_m)
      movel([0.274158, -1.413138, -2.545696, -0.753555, 1.570796, 1.844954],accel_mss,speed_ms,0,blend_radius_m)
      movel([0.273733, -1.414913, -2.544356, -0.753121, 1.570796, 1.844530],accel_mss,speed_ms,0,blend_radius_m)
      movel([0.273339, -1.416677, -2.543018, -0.752694, 1.570796, 1.844136],accel_mss,speed_ms,0,blend_radius_m)
      movel([0.273190, -1.417438, -2.542440, -0.752511, 1.570796, 1.843987],accel_mss,speed_ms,0,blend_radius_m)
      movel([0.273073, -1.418191, -2.541867, -0.752331, 1.570796, 1.843869],accel_mss,speed_ms,0,blend_radius_m)
      movel([0.272984, -1.418937, -2.541298, -0.752153, 1.570796, 1.843780],accel_mss,speed_ms,0,blend_radius_m)
      movel([0.272921, -1.419692, -2.540722, -0.751974, 1.570796, 1.843718],accel_mss,speed_ms,0,blend_radius_m)
      movel([0.272881, -1.420440, -2.540151, -0.751798, 1.570796, 1.843677],accel_mss,speed_ms,0,blend_radius_m)
      movel([0.272867, -1.421180, -2.539585, -0.751625, 1.570796, 1.843663],accel_mss,speed_ms,0,blend_radius_m)
      movel([0.272876, -1.421910, -2.539025, -0.751454, 1.570796, 1.843672],accel_mss,speed_ms,0,blend_radius_m)
      movel([0.272907, -1.422631, -2.538471, -0.751286, 1.570796, 1.843703],accel_mss,speed_ms,0,blend_radius_m)
      movel([0.272962, -1.423345, -2.537923, -0.751121, 1.570796, 1.843759],accel_mss,speed_ms,0,blend_radius_m)
      movel([0.273044, -1.424045, -2.537384, -0.750960, 1.570796, 1.843840],accel_mss,speed_ms,0,blend_radius_m)
      movel([0.273146, -1.424735, -2.536852, -0.750802, 1.570796, 1.843942],accel_mss,speed_ms,0,blend_radius_m)
      movel([0.273277, -1.425445, -2.536304, -0.750640, 1.570796, 1.844073],accel_mss,speed_ms,0,blend_radius_m)
      movel([0.273430, -1.426145, -2.535763, -0.750481, 1.570796, 1.844226],accel_mss,speed_ms,0,blend_radius_m)
      movel([0.273602, -1.426833, -2.535231, -0.750325, 1.570796, 1.844399],accel_mss,speed_ms,0,blend_radius_m)
      movel([0.273797, -1.427509, -2.534707, -0.750173, 1.570796, 1.844594],accel_mss,speed_ms,0,blend_radius_m)
      movel([0.274010, -1.428175, -2.534190, -0.750024, 1.570796, 1.844807],accel_mss,speed_ms,0,blend_radius_m)
      movel([0.274246, -1.428829, -2.533682, -0.749878, 1.570796, 1.845043],accel_mss,speed_ms,0,blend_radius_m)
      movel([0.274502, -1.429469, -2.533184, -0.749736, 1.570796, 1.845298],accel_mss,speed_ms,0,blend_radius_m)
      movel([0.274780, -1.430099, -2.532694, -0.749597, 1.570796, 1.845576],accel_mss,speed_ms,0,blend_radius_m)
      movel([0.275084, -1.430733, -2.532199, -0.749457, 1.570796, 1.845880],accel_mss,speed_ms,0,blend_radius_m)
      movel([0.275409, -1.431356, -2.531713, -0.749320, 1.570796, 1.846205],accel_mss,speed_ms,0,blend_radius_m)
      movel([0.275752, -1.431965, -2.531236, -0.749187, 1.570796, 1.846549],accel_mss,speed_ms,0,blend_radius_m)
      movel([0.276118, -1.432560, -2.530771, -0.749058, 1.570796, 1.846914],accel_mss,speed_ms,0,blend_radius_m)
      movel([0.276502, -1.433140, -2.530317, -0.748932, 1.570796, 1.847298],accel_mss,speed_ms,0,blend_radius_m)
      movel([0.276903, -1.433708, -2.529871, -0.748810, 1.570796, 1.847699],accel_mss,speed_ms,0,blend_radius_m)
      movel([0.277325, -1.434260, -2.529438, -0.748691, 1.570796, 1.848122],accel_mss,speed_ms,0,blend_radius_m)
      movel([0.277765, -1.434798, -2.529015, -0.748576, 1.570796, 1.848561],accel_mss,speed_ms,0,blend_radius_m)
      movel([0.278226, -1.435332, -2.528595, -0.748462, 1.570796, 1.849023],accel_mss,speed_ms,0,blend_radius_m)
      movel([0.278709, -1.435847, -2.528189, -0.748353, 1.570796, 1.849505],accel_mss,speed_ms,0,blend_radius_m)
      movel([0.279207, -1.436351, -2.527792, -0.748246, 1.570796, 1.850003],accel_mss,speed_ms,0,blend_radius_m)
      movel([0.279723, -1.436837, -2.527408, -0.748144, 1.570796, 1.850519],accel_mss,speed_ms,0,blend_radius_m)
      movel([0.280256, -1.437309, -2.527035, -0.748045, 1.570796, 1.851052],accel_mss,speed_ms,0,blend_radius_m)
      movel([0.280804, -1.437766, -2.526674, -0.747949, 1.570796, 1.851600],accel_mss,speed_ms,0,blend_radius_m)
      movel([0.281369, -1.438207, -2.526325, -0.747857, 1.570796, 1.852166],accel_mss,speed_ms,0,blend_radius_m)
      movel([0.281949, -1.438633, -2.525987, -0.747768, 1.570796, 1.852746],accel_mss,speed_ms,0,blend_radius_m)
      movel([0.282588, -1.439072, -2.525640, -0.747677, 1.570796, 1.853385],accel_mss,speed_ms,0,blend_radius_m)
      movel([0.283242, -1.439496, -2.525304, -0.747589, 1.570796, 1.854038],accel_mss,speed_ms,0,blend_radius_m)
      movel([0.283914, -1.439900, -2.524983, -0.747506, 1.570796, 1.854711],accel_mss,speed_ms,0,blend_radius_m)
      movel([0.284599, -1.440289, -2.524674, -0.747426, 1.570796, 1.855395],accel_mss,speed_ms,0,blend_radius_m)
      movel([0.285300, -1.440660, -2.524379, -0.747350, 1.570796, 1.856097],accel_mss,speed_ms,0,blend_radius_m)
      movel([0.286016, -1.441015, -2.524097, -0.747278, 1.570796, 1.856813],accel_mss,speed_ms,0,blend_radius_m)
      movel([0.286747, -1.441351, -2.523829, -0.747209, 1.570796, 1.857543],accel_mss,speed_ms,0,blend_radius_m)
      movel([0.287491, -1.441669, -2.523576, -0.747144, 1.570796, 1.858287],accel_mss,speed_ms,0,blend_radius_m)
      movel([0.288283, -1.441985, -2.523324, -0.747080, 1.570796, 1.859079],accel_mss,speed_ms,0,blend_radius_m)
      movel([0.289086, -1.442285, -2.523085, -0.747020, 1.570796, 1.859882],accel_mss,speed_ms,0,blend_radius_m)
      movel([0.289902, -1.442568, -2.522859, -0.746962, 1.570796, 1.860699],accel_mss,speed_ms,0,blend_radius_m)
      movel([0.290730, -1.442835, -2.522646, -0.746909, 1.570796, 1.861526],accel_mss,speed_ms,0,blend_radius_m)
      movel([0.291569, -1.443085, -2.522446, -0.746858, 1.570796, 1.862365],accel_mss,speed_ms,0,blend_radius_m)
      movel([0.292422, -1.443317, -2.522260, -0.746811, 1.570796, 1.863218],accel_mss,speed_ms,0,blend_radius_m)
      movel([0.293283, -1.443535, -2.522086, -0.746768, 1.570796, 1.864079],accel_mss,speed_ms,0,blend_radius_m)
      movel([0.294154, -1.443735, -2.521926, -0.746728, 1.570796, 1.864951],accel_mss,speed_ms,0,blend_radius_m)
      movel([0.295057, -1.443924, -2.521775, -0.746690, 1.570796, 1.865853],accel_mss,speed_ms,0,blend_radius_m)
      movel([0.295971, -1.444096, -2.521637, -0.746656, 1.570796, 1.866767],accel_mss,speed_ms,0,blend_radius_m)
      movel([0.296894, -1.444252, -2.521512, -0.746625, 1.570796, 1.867690],accel_mss,speed_ms,0,blend_radius_m)
      movel([0.297825, -1.444391, -2.521401, -0.746597, 1.570796, 1.868621],accel_mss,speed_ms,0,blend_radius_m)
      movel([0.298768, -1.444511, -2.521305, -0.746573, 1.570796, 1.869564],accel_mss,speed_ms,0,blend_radius_m)
      movel([0.299720, -1.444616, -2.521221, -0.746552, 1.570796, 1.870516],accel_mss,speed_ms,0,blend_radius_m)
      movel([0.300679, -1.444705, -2.521150, -0.746534, 1.570796, 1.871476],accel_mss,speed_ms,0,blend_radius_m)
      movel([0.301647, -1.444776, -2.521092, -0.746520, 1.570796, 1.872443],accel_mss,speed_ms,0,blend_radius_m)
      movel([0.302623, -1.444832, -2.521048, -0.746509, 1.570796, 1.873420],accel_mss,speed_ms,0,blend_radius_m)
      movel([0.303608, -1.444870, -2.521017, -0.746502, 1.570796, 1.874404],accel_mss,speed_ms,0,blend_radius_m)
      movel([0.304602, -1.444890, -2.521001, -0.746498, 1.570796, 1.875399],accel_mss,speed_ms,0,blend_radius_m)
      movel([0.305600, -1.444895, -2.520997, -0.746497, 1.570796, 1.876396],accel_mss,speed_ms,0,blend_radius_m)
      movel([0.306608, -1.444882, -2.521008, -0.746499, 1.570796, 1.877404],accel_mss,speed_ms,0,blend_radius_m)
      movel([0.307621, -1.444853, -2.521031, -0.746505, 1.570796, 1.878418],accel_mss,speed_ms,0,blend_radius_m)
      movel([0.308643, -1.444807, -2.521068, -0.746514, 1.570796, 1.879439],accel_mss,speed_ms,0,blend_radius_m)
      movel([0.309668, -1.444744, -2.521118, -0.746527, 1.570796, 1.880464],accel_mss,speed_ms,0,blend_radius_m)
      movel([0.312678, -1.444539, -2.521282, -0.746567, 1.570796, 1.883474],accel_mss,speed_ms,0,blend_radius_m)
      movel([0.312279, -1.445688, -2.520361, -0.746340, 1.570796, 1.883075],accel_mss,speed_ms,0,blend_radius_m)
      movel([0.311880, -1.446834, -2.519440, -0.746115, 1.570796, 1.882677],accel_mss,speed_ms,0,blend_radius_m)
      movel([0.280216, -1.449370, -2.517394, -0.745625, 1.570796, 1.851012],accel_mss,speed_ms,0,blend_radius_m)
      movel([0.248377, -1.452781, -2.514627, -0.744981, 1.570796, 1.819173],accel_mss,speed_ms,0,blend_radius_m)
      movel([0.259911, -1.412348, -2.546291, -0.753750, 1.570796, 1.830707],accel_mss,speed_ms,0,blend_radius_m)
      movel([0.272608, -1.369235, -2.577388, -0.765765, 1.570796, 1.843404],accel_mss,speed_ms,0,blend_radius_m)
      movel([0.307596, -1.364998, -2.580301, -0.767090, 1.570796, 1.878392],accel_mss,speed_ms,0,blend_radius_m)
      movel([0.342353, -1.361839, -2.582456, -0.768095, 1.570796, 1.913150],accel_mss,speed_ms,0,blend_radius_m)
      speed_ms = 0.003
      movel([0.342353, -1.365171, -2.583973, -0.763245, 1.570796, 1.913150],accel_mss,speed_ms,0,blend_radius_m)
      speed_ms = 0.007
      movel([0.341641, -1.367098, -2.582653, -0.762638, 1.570796, 1.912437],accel_mss,speed_ms,0,blend_radius_m)
      movel([0.340931, -1.369019, -2.581333, -0.762037, 1.570796, 1.911728],accel_mss,speed_ms,0,blend_radius_m)
      movel([0.336123, -1.369495, -2.581005, -0.761889, 1.570796, 1.906919],accel_mss,speed_ms,0,blend_radius_m)
      movel([0.334430, -1.369677, -2.580880, -0.761833, 1.570796, 1.905226],accel_mss,speed_ms,0,blend_radius_m)
      movel([0.332727, -1.369882, -2.580738, -0.761769, 1.570796, 1.903523],accel_mss,speed_ms,0,blend_radius_m)
      movel([0.331393, -1.370071, -2.580608, -0.761710, 1.570796, 1.902189],accel_mss,speed_ms,0,blend_radius_m)
      movel([0.330047, -1.370293, -2.580454, -0.761642, 1.570796, 1.900843],accel_mss,speed_ms,0,blend_radius_m)
      movel([0.328764, -1.370539, -2.580285, -0.761566, 1.570796, 1.899560],accel_mss,speed_ms,0,blend_radius_m)
      movel([0.327473, -1.370819, -2.580091, -0.761479, 1.570796, 1.898270],accel_mss,speed_ms,0,blend_radius_m)
      movel([0.325956, -1.371181, -2.579840, -0.761367, 1.570796, 1.896752],accel_mss,speed_ms,0,blend_radius_m)
      movel([0.324433, -1.371572, -2.579570, -0.761247, 1.570796, 1.895230],accel_mss,speed_ms,0,blend_radius_m)
      movel([0.323162, -1.371918, -2.579330, -0.761141, 1.570796, 1.893958],accel_mss,speed_ms,0,blend_radius_m)
      movel([0.321888, -1.372291, -2.579072, -0.761026, 1.570796, 1.892684],accel_mss,speed_ms,0,blend_radius_m)
      movel([0.320612, -1.372686, -2.578798, -0.760905, 1.570796, 1.891408],accel_mss,speed_ms,0,blend_radius_m)
      movel([0.319335, -1.373106, -2.578506, -0.760777, 1.570796, 1.890132],accel_mss,speed_ms,0,blend_radius_m)
      movel([0.318059, -1.373549, -2.578198, -0.760642, 1.570796, 1.888855],accel_mss,speed_ms,0,blend_radius_m)
      movel([0.316792, -1.374012, -2.577876, -0.760501, 1.570796, 1.887588],accel_mss,speed_ms,0,blend_radius_m)
      movel([0.315526, -1.374498, -2.577538, -0.760353, 1.570796, 1.886322],accel_mss,speed_ms,0,blend_radius_m)
      movel([0.314261, -1.375009, -2.577181, -0.760198, 1.570796, 1.885058],accel_mss,speed_ms,0,blend_radius_m)
      movel([0.312998, -1.375541, -2.576811, -0.760037, 1.570796, 1.883794],accel_mss,speed_ms,0,blend_radius_m)
      movel([0.311739, -1.376095, -2.576424, -0.759870, 1.570796, 1.882536],accel_mss,speed_ms,0,blend_radius_m)
      movel([0.310506, -1.376662, -2.576027, -0.759700, 1.570796, 1.881302],accel_mss,speed_ms,0,blend_radius_m)
      movel([0.309278, -1.377249, -2.575616, -0.759524, 1.570796, 1.880074],accel_mss,speed_ms,0,blend_radius_m)
      movel([0.308056, -1.377858, -2.575189, -0.759342, 1.570796, 1.878852],accel_mss,speed_ms,0,blend_radius_m)
      movel([0.306839, -1.378489, -2.574747, -0.759153, 1.570796, 1.877635],accel_mss,speed_ms,0,blend_radius_m)
      movel([0.305626, -1.379139, -2.574290, -0.758960, 1.570796, 1.876423],accel_mss,speed_ms,0,blend_radius_m)
      movel([0.304459, -1.379790, -2.573832, -0.758767, 1.570796, 1.875255],accel_mss,speed_ms,0,blend_radius_m)
      movel([0.303297, -1.380464, -2.573357, -0.758568, 1.570796, 1.874093],accel_mss,speed_ms,0,blend_radius_m)
      movel([0.302144, -1.381155, -2.572869, -0.758365, 1.570796, 1.872941],accel_mss,speed_ms,0,blend_radius_m)
      movel([0.301002, -1.381868, -2.572365, -0.758155, 1.570796, 1.871798],accel_mss,speed_ms,0,blend_radius_m)
      movel([0.299869, -1.382599, -2.571848, -0.757942, 1.570796, 1.870665],accel_mss,speed_ms,0,blend_radius_m)
      movel([0.299135, -1.383092, -2.571498, -0.757798, 1.570796, 1.869931],accel_mss,speed_ms,0,blend_radius_m)
      movel([0.298406, -1.383599, -2.571139, -0.757651, 1.570796, 1.869202],accel_mss,speed_ms,0,blend_radius_m)
      movel([0.297686, -1.384117, -2.570771, -0.757501, 1.570796, 1.868482],accel_mss,speed_ms,0,blend_radius_m)
      movel([0.296342, -1.385117, -2.570060, -0.757212, 1.570796, 1.867138],accel_mss,speed_ms,0,blend_radius_m)
      movel([0.295013, -1.386134, -2.569336, -0.756919, 1.570796, 1.865810],accel_mss,speed_ms,0,blend_radius_m)
      movel([0.293697, -1.387171, -2.568595, -0.756623, 1.570796, 1.864493],accel_mss,speed_ms,0,blend_radius_m)
      movel([0.292396, -1.388222, -2.567843, -0.756324, 1.570796, 1.863193],accel_mss,speed_ms,0,blend_radius_m)
      movel([0.291708, -1.388794, -2.567433, -0.756162, 1.570796, 1.862504],accel_mss,speed_ms,0,blend_radius_m)
      movel([0.291033, -1.389377, -2.567015, -0.755997, 1.570796, 1.861829],accel_mss,speed_ms,0,blend_radius_m)
      movel([0.290369, -1.389969, -2.566590, -0.755831, 1.570796, 1.861165],accel_mss,speed_ms,0,blend_radius_m)
      movel([0.289528, -1.390743, -2.566032, -0.755613, 1.570796, 1.860324],accel_mss,speed_ms,0,blend_radius_m)
      movel([0.288705, -1.391528, -2.565467, -0.755394, 1.570796, 1.859502],accel_mss,speed_ms,0,blend_radius_m)
      movel([0.287899, -1.392323, -2.564893, -0.755173, 1.570796, 1.858695],accel_mss,speed_ms,0,blend_radius_m)
      movel([0.287109, -1.393129, -2.564311, -0.754949, 1.570796, 1.857905],accel_mss,speed_ms,0,blend_radius_m)
      movel([0.286337, -1.393945, -2.563720, -0.754724, 1.570796, 1.857133],accel_mss,speed_ms,0,blend_radius_m)
      movel([0.285582, -1.394768, -2.563123, -0.754498, 1.570796, 1.856378],accel_mss,speed_ms,0,blend_radius_m)
      movel([0.284855, -1.395592, -2.562524, -0.754273, 1.570796, 1.855651],accel_mss,speed_ms,0,blend_radius_m)
      movel([0.284146, -1.396422, -2.561921, -0.754047, 1.570796, 1.854942],accel_mss,speed_ms,0,blend_radius_m)
      movel([0.283459, -1.397260, -2.561309, -0.753819, 1.570796, 1.854256],accel_mss,speed_ms,0,blend_radius_m)
      movel([0.282791, -1.398105, -2.560693, -0.753591, 1.570796, 1.853587],accel_mss,speed_ms,0,blend_radius_m)
      movel([0.282143, -1.398956, -2.560070, -0.753363, 1.570796, 1.852939],accel_mss,speed_ms,0,blend_radius_m)
      movel([0.281518, -1.399813, -2.559442, -0.753134, 1.570796, 1.852314],accel_mss,speed_ms,0,blend_radius_m)
      movel([0.280925, -1.400656, -2.558823, -0.752909, 1.570796, 1.851721],accel_mss,speed_ms,0,blend_radius_m)
      movel([0.280356, -1.401505, -2.558200, -0.752685, 1.570796, 1.851152],accel_mss,speed_ms,0,blend_radius_m)
      movel([0.279807, -1.402358, -2.557572, -0.752460, 1.570796, 1.850603],accel_mss,speed_ms,0,blend_radius_m)
      movel([0.279280, -1.403212, -2.556942, -0.752236, 1.570796, 1.850077],accel_mss,speed_ms,0,blend_radius_m)
      movel([0.278776, -1.404070, -2.556307, -0.752011, 1.570796, 1.849572],accel_mss,speed_ms,0,blend_radius_m)
      movel([0.278297, -1.404929, -2.555671, -0.751788, 1.570796, 1.849094],accel_mss,speed_ms,0,blend_radius_m)
      movel([0.277915, -1.405646, -2.555140, -0.751603, 1.570796, 1.848711],accel_mss,speed_ms,0,blend_radius_m)
      movel([0.277553, -1.406364, -2.554607, -0.751418, 1.570796, 1.848349],accel_mss,speed_ms,0,blend_radius_m)
      movel([0.277207, -1.407084, -2.554072, -0.751233, 1.570796, 1.848003],accel_mss,speed_ms,0,blend_radius_m)
      movel([0.276882, -1.407800, -2.553539, -0.751050, 1.570796, 1.847679],accel_mss,speed_ms,0,blend_radius_m)
      movel([0.276573, -1.408518, -2.553003, -0.750867, 1.570796, 1.847370],accel_mss,speed_ms,0,blend_radius_m)
      movel([0.276285, -1.409235, -2.552468, -0.750686, 1.570796, 1.847081],accel_mss,speed_ms,0,blend_radius_m)
      movel([0.276016, -1.409949, -2.551934, -0.750506, 1.570796, 1.846812],accel_mss,speed_ms,0,blend_radius_m)
      movel([0.275694, -1.410866, -2.551248, -0.750275, 1.570796, 1.846490],accel_mss,speed_ms,0,blend_radius_m)
      movel([0.275399, -1.411776, -2.550565, -0.750048, 1.570796, 1.846196],accel_mss,speed_ms,0,blend_radius_m)
      movel([0.275130, -1.412684, -2.549882, -0.749822, 1.570796, 1.845926],accel_mss,speed_ms,0,blend_radius_m)
      movel([0.274626, -1.414511, -2.548505, -0.749372, 1.570796, 1.845423],accel_mss,speed_ms,0,blend_radius_m)
      movel([0.274158, -1.416330, -2.547130, -0.748929, 1.570796, 1.844954],accel_mss,speed_ms,0,blend_radius_m)
      movel([0.273733, -1.418100, -2.545787, -0.748503, 1.570796, 1.844530],accel_mss,speed_ms,0,blend_radius_m)
      movel([0.273339, -1.419859, -2.544447, -0.748083, 1.570796, 1.844136],accel_mss,speed_ms,0,blend_radius_m)
      movel([0.273190, -1.420618, -2.543867, -0.747904, 1.570796, 1.843987],accel_mss,speed_ms,0,blend_radius_m)
      movel([0.273073, -1.421368, -2.543293, -0.747727, 1.570796, 1.843869],accel_mss,speed_ms,0,blend_radius_m)
      movel([0.272984, -1.422113, -2.542723, -0.747553, 1.570796, 1.843780],accel_mss,speed_ms,0,blend_radius_m)
      movel([0.272921, -1.422866, -2.542146, -0.747378, 1.570796, 1.843718],accel_mss,speed_ms,0,blend_radius_m)
      movel([0.272881, -1.423611, -2.541573, -0.747205, 1.570796, 1.843677],accel_mss,speed_ms,0,blend_radius_m)
      movel([0.272867, -1.424349, -2.541006, -0.747034, 1.570796, 1.843663],accel_mss,speed_ms,0,blend_radius_m)
      movel([0.272876, -1.425077, -2.540445, -0.746867, 1.570796, 1.843672],accel_mss,speed_ms,0,blend_radius_m)
      movel([0.272907, -1.425796, -2.539890, -0.746703, 1.570796, 1.843703],accel_mss,speed_ms,0,blend_radius_m)
      movel([0.272962, -1.426507, -2.539341, -0.746541, 1.570796, 1.843759],accel_mss,speed_ms,0,blend_radius_m)
      movel([0.273044, -1.427205, -2.538801, -0.746383, 1.570796, 1.843840],accel_mss,speed_ms,0,blend_radius_m)
      movel([0.273146, -1.427894, -2.538267, -0.746227, 1.570796, 1.843942],accel_mss,speed_ms,0,blend_radius_m)
      movel([0.273277, -1.428602, -2.537719, -0.746069, 1.570796, 1.844073],accel_mss,speed_ms,0,blend_radius_m)
      movel([0.273430, -1.429300, -2.537176, -0.745913, 1.570796, 1.844226],accel_mss,speed_ms,0,blend_radius_m)
      movel([0.273602, -1.429985, -2.536643, -0.745760, 1.570796, 1.844399],accel_mss,speed_ms,0,blend_radius_m)
      movel([0.273797, -1.430660, -2.536118, -0.745611, 1.570796, 1.844594],accel_mss,speed_ms,0,blend_radius_m)
      movel([0.274010, -1.431323, -2.535601, -0.745465, 1.570796, 1.844807],accel_mss,speed_ms,0,blend_radius_m)
      movel([0.274246, -1.431976, -2.535091, -0.745322, 1.570796, 1.845043],accel_mss,speed_ms,0,blend_radius_m)
      movel([0.274502, -1.432615, -2.534592, -0.745183, 1.570796, 1.845298],accel_mss,speed_ms,0,blend_radius_m)
      movel([0.274780, -1.433242, -2.534101, -0.745046, 1.570796, 1.845576],accel_mss,speed_ms,0,blend_radius_m)
      movel([0.275084, -1.433874, -2.533605, -0.744909, 1.570796, 1.845880],accel_mss,speed_ms,0,blend_radius_m)
      movel([0.275409, -1.434496, -2.533118, -0.744775, 1.570796, 1.846205],accel_mss,speed_ms,0,blend_radius_m)
      movel([0.275752, -1.435103, -2.532641, -0.744645, 1.570796, 1.846549],accel_mss,speed_ms,0,blend_radius_m)
      movel([0.276118, -1.435696, -2.532174, -0.744519, 1.570796, 1.846914],accel_mss,speed_ms,0,blend_radius_m)
      movel([0.276502, -1.436275, -2.531719, -0.744396, 1.570796, 1.847298],accel_mss,speed_ms,0,blend_radius_m)
      movel([0.276903, -1.436841, -2.531272, -0.744276, 1.570796, 1.847699],accel_mss,speed_ms,0,blend_radius_m)
      movel([0.277325, -1.437391, -2.530838, -0.744159, 1.570796, 1.848122],accel_mss,speed_ms,0,blend_radius_m)
      movel([0.277765, -1.437928, -2.530415, -0.744047, 1.570796, 1.848561],accel_mss,speed_ms,0,blend_radius_m)
      movel([0.278226, -1.438460, -2.529994, -0.743935, 1.570796, 1.849023],accel_mss,speed_ms,0,blend_radius_m)
      movel([0.278709, -1.438974, -2.529587, -0.743828, 1.570796, 1.849505],accel_mss,speed_ms,0,blend_radius_m)
      movel([0.279207, -1.439476, -2.529189, -0.743724, 1.570796, 1.850003],accel_mss,speed_ms,0,blend_radius_m)
      movel([0.279723, -1.439960, -2.528805, -0.743624, 1.570796, 1.850519],accel_mss,speed_ms,0,blend_radius_m)
      movel([0.280256, -1.440431, -2.528431, -0.743526, 1.570796, 1.851052],accel_mss,speed_ms,0,blend_radius_m)
      movel([0.280804, -1.440887, -2.528069, -0.743433, 1.570796, 1.851600],accel_mss,speed_ms,0,blend_radius_m)
      movel([0.281369, -1.441327, -2.527719, -0.743343, 1.570796, 1.852166],accel_mss,speed_ms,0,blend_radius_m)
      movel([0.281949, -1.441752, -2.527381, -0.743256, 1.570796, 1.852746],accel_mss,speed_ms,0,blend_radius_m)
      movel([0.282588, -1.442190, -2.527033, -0.743167, 1.570796, 1.853385],accel_mss,speed_ms,0,blend_radius_m)
      movel([0.283242, -1.442612, -2.526696, -0.743081, 1.570796, 1.854038],accel_mss,speed_ms,0,blend_radius_m)
      movel([0.283914, -1.443015, -2.526375, -0.742999, 1.570796, 1.854711],accel_mss,speed_ms,0,blend_radius_m)
      movel([0.284599, -1.443403, -2.526065, -0.742921, 1.570796, 1.855395],accel_mss,speed_ms,0,blend_radius_m)
      movel([0.285300, -1.443772, -2.525770, -0.742847, 1.570796, 1.856097],accel_mss,speed_ms,0,blend_radius_m)
      movel([0.286016, -1.444127, -2.525487, -0.742776, 1.570796, 1.856813],accel_mss,speed_ms,0,blend_radius_m)
      movel([0.286747, -1.444462, -2.525218, -0.742709, 1.570796, 1.857543],accel_mss,speed_ms,0,blend_radius_m)
      movel([0.287491, -1.444779, -2.524965, -0.742646, 1.570796, 1.858287],accel_mss,speed_ms,0,blend_radius_m)
      movel([0.288283, -1.445094, -2.524712, -0.742583, 1.570796, 1.859079],accel_mss,speed_ms,0,blend_radius_m)
      movel([0.289086, -1.445393, -2.524473, -0.742524, 1.570796, 1.859882],accel_mss,speed_ms,0,blend_radius_m)
      movel([0.289902, -1.445675, -2.524246, -0.742468, 1.570796, 1.860699],accel_mss,speed_ms,0,blend_radius_m)
      movel([0.290730, -1.445941, -2.524033, -0.742415, 1.570796, 1.861526],accel_mss,speed_ms,0,blend_radius_m)
      movel([0.291569, -1.446191, -2.523832, -0.742366, 1.570796, 1.862365],accel_mss,speed_ms,0,blend_radius_m)
      movel([0.292422, -1.446422, -2.523647, -0.742320, 1.570796, 1.863218],accel_mss,speed_ms,0,blend_radius_m)
      movel([0.293283, -1.446640, -2.523472, -0.742277, 1.570796, 1.864079],accel_mss,speed_ms,0,blend_radius_m)
      movel([0.294154, -1.446839, -2.523312, -0.742238, 1.570796, 1.864951],accel_mss,speed_ms,0,blend_radius_m)
      movel([0.295057, -1.447027, -2.523161, -0.742201, 1.570796, 1.865853],accel_mss,speed_ms,0,blend_radius_m)
      movel([0.295971, -1.447198, -2.523023, -0.742168, 1.570796, 1.866767],accel_mss,speed_ms,0,blend_radius_m)
      movel([0.296894, -1.447354, -2.522897, -0.742137, 1.570796, 1.867690],accel_mss,speed_ms,0,blend_radius_m)
      movel([0.297825, -1.447492, -2.522786, -0.742110, 1.570796, 1.868621],accel_mss,speed_ms,0,blend_radius_m)
      movel([0.298768, -1.447613, -2.522689, -0.742087, 1.570796, 1.869564],accel_mss,speed_ms,0,blend_radius_m)
      movel([0.299720, -1.447717, -2.522605, -0.742067, 1.570796, 1.870516],accel_mss,speed_ms,0,blend_radius_m)
      movel([0.300679, -1.447806, -2.522534, -0.742049, 1.570796, 1.871476],accel_mss,speed_ms,0,blend_radius_m)
      movel([0.301647, -1.447877, -2.522476, -0.742036, 1.570796, 1.872443],accel_mss,speed_ms,0,blend_radius_m)
      movel([0.302623, -1.447932, -2.522432, -0.742025, 1.570796, 1.873420],accel_mss,speed_ms,0,blend_radius_m)
      movel([0.303608, -1.447970, -2.522401, -0.742017, 1.570796, 1.874404],accel_mss,speed_ms,0,blend_radius_m)
      movel([0.304602, -1.447990, -2.522385, -0.742014, 1.570796, 1.875399],accel_mss,speed_ms,0,blend_radius_m)
      movel([0.305600, -1.447995, -2.522381, -0.742013, 1.570796, 1.876396],accel_mss,speed_ms,0,blend_radius_m)
      movel([0.306608, -1.447982, -2.522392, -0.742015, 1.570796, 1.877404],accel_mss,speed_ms,0,blend_radius_m)
      movel([0.307621, -1.447954, -2.522415, -0.742021, 1.570796, 1.878418],accel_mss,speed_ms,0,blend_radius_m)
      movel([0.308643, -1.447908, -2.522452, -0.742030, 1.570796, 1.879439],accel_mss,speed_ms,0,blend_radius_m)
      movel([0.309668, -1.447845, -2.522503, -0.742042, 1.570796, 1.880464],accel_mss,speed_ms,0,blend_radius_m)
      movel([0.312678, -1.447641, -2.522667, -0.742082, 1.570796, 1.883474],accel_mss,speed_ms,0,blend_radius_m)
      movel([0.312279, -1.448786, -2.521744, -0.741859, 1.570796, 1.883075],accel_mss,speed_ms,0,blend_radius_m)
      movel([0.311880, -1.449928, -2.520821, -0.741640, 1.570796, 1.882677],accel_mss,speed_ms,0,blend_radius_m)
      movel([0.280216, -1.452458, -2.518771, -0.741161, 1.570796, 1.851012],accel_mss,speed_ms,0,blend_radius_m)
      movel([0.248377, -1.455858, -2.515999, -0.740532, 1.570796, 1.819173],accel_mss,speed_ms,0,blend_radius_m)
      movel([0.259911, -1.415542, -2.547726, -0.749121, 1.570796, 1.830707],accel_mss,speed_ms,0,blend_radius_m)
      movel([0.272608, -1.372548, -2.578894, -0.760948, 1.570796, 1.843404],accel_mss,speed_ms,0,blend_radius_m)
      movel([0.307596, -1.368321, -2.581813, -0.762255, 1.570796, 1.878392],accel_mss,speed_ms,0,blend_radius_m)
      movel([0.342353, -1.365171, -2.583973, -0.763245, 1.570796, 1.913150],accel_mss,speed_ms,0,blend_radius_m)
      speed_ms = 0.003
      movel([0.342353, -1.351985, -2.577853, -0.782552, 1.570796, 1.913150],accel_mss,speed_ms,0,blend_radius_m)
      speed_ms = 0.01
      movel([0.342353, -1.326735, -2.565220, -0.820435, 1.570796, 1.913150],accel_mss,speed_ms,0,blend_radius_m)
      movel([0.338485, -1.335837, -2.559287, -0.817264, 1.570796, 1.909281],accel_mss,speed_ms,0,blend_radius_m)
      movel([0.338485, -1.360932, -2.571804, -0.779653, 1.570796, 1.909281],accel_mss,speed_ms,0,blend_radius_m)
      speed_ms = 0.003
      movel([0.338485, -1.370719, -2.576362, -0.765307, 1.570796, 1.909281],accel_mss,speed_ms,0,blend_radius_m)
      speed_ms = 0.007
      movel([0.338879, -1.370800, -2.576307, -0.765283, 1.570796, 1.909676],accel_mss,speed_ms,0,blend_radius_m)
      movel([0.326050, -1.405916, -2.551102, -0.755371, 1.570796, 1.896846],accel_mss,speed_ms,0,blend_radius_m)
      movel([0.321364, -1.418935, -2.541300, -0.752154, 1.570796, 1.892160],accel_mss,speed_ms,0,blend_radius_m)
      movel([0.317469, -1.429815, -2.532915, -0.749659, 1.570796, 1.888265],accel_mss,speed_ms,0,blend_radius_m)
      movel([0.314074, -1.439350, -2.525419, -0.747620, 1.570796, 1.884870],accel_mss,speed_ms,0,blend_radius_m)
      movel([0.313964, -1.439634, -2.525194, -0.747561, 1.570796, 1.884760],accel_mss,speed_ms,0,blend_radius_m)
      movel([0.313839, -1.439917, -2.524969, -0.747503, 1.570796, 1.884635],accel_mss,speed_ms,0,blend_radius_m)
      movel([0.313503, -1.440625, -2.524406, -0.747357, 1.570796, 1.884299],accel_mss,speed_ms,0,blend_radius_m)
      movel([0.310537, -1.440829, -2.524244, -0.747315, 1.570796, 1.881334],accel_mss,speed_ms,0,blend_radius_m)
      movel([0.309649, -1.440886, -2.524199, -0.747304, 1.570796, 1.880445],accel_mss,speed_ms,0,blend_radius_m)
      movel([0.308768, -1.440926, -2.524167, -0.747296, 1.570796, 1.879564],accel_mss,speed_ms,0,blend_radius_m)
      movel([0.307891, -1.440955, -2.524144, -0.747290, 1.570796, 1.878688],accel_mss,speed_ms,0,blend_radius_m)
      movel([0.307019, -1.440970, -2.524132, -0.747287, 1.570796, 1.877816],accel_mss,speed_ms,0,blend_radius_m)
      movel([0.306154, -1.440972, -2.524131, -0.747286, 1.570796, 1.876950],accel_mss,speed_ms,0,blend_radius_m)
      movel([0.305293, -1.440961, -2.524139, -0.747288, 1.570796, 1.876089],accel_mss,speed_ms,0,blend_radius_m)
      movel([0.304439, -1.440935, -2.524160, -0.747294, 1.570796, 1.875235],accel_mss,speed_ms,0,blend_radius_m)
      movel([0.303591, -1.440897, -2.524190, -0.747302, 1.570796, 1.874388],accel_mss,speed_ms,0,blend_radius_m)
      movel([0.302750, -1.440845, -2.524232, -0.747312, 1.570796, 1.873547],accel_mss,speed_ms,0,blend_radius_m)
      movel([0.301914, -1.440779, -2.524284, -0.747326, 1.570796, 1.872710],accel_mss,speed_ms,0,blend_radius_m)
      movel([0.301086, -1.440700, -2.524347, -0.747342, 1.570796, 1.871882],accel_mss,speed_ms,0,blend_radius_m)
      movel([0.300266, -1.440608, -2.524420, -0.747361, 1.570796, 1.871063],accel_mss,speed_ms,0,blend_radius_m)
      movel([0.299452, -1.440500, -2.524506, -0.747383, 1.570796, 1.870248],accel_mss,speed_ms,0,blend_radius_m)
      movel([0.298658, -1.440384, -2.524599, -0.747407, 1.570796, 1.869454],accel_mss,speed_ms,0,blend_radius_m)
      movel([0.297871, -1.440251, -2.524704, -0.747434, 1.570796, 1.868667],accel_mss,speed_ms,0,blend_radius_m)
      movel([0.297094, -1.440106, -2.524819, -0.747464, 1.570796, 1.867890],accel_mss,speed_ms,0,blend_radius_m)
      movel([0.296324, -1.439945, -2.524947, -0.747497, 1.570796, 1.867120],accel_mss,speed_ms,0,blend_radius_m)
      movel([0.295562, -1.439772, -2.525084, -0.747532, 1.570796, 1.866359],accel_mss,speed_ms,0,blend_radius_m)
      movel([0.294809, -1.439587, -2.525231, -0.747571, 1.570796, 1.865605],accel_mss,speed_ms,0,blend_radius_m)
      movel([0.294067, -1.439385, -2.525391, -0.747612, 1.570796, 1.864863],accel_mss,speed_ms,0,blend_radius_m)
      movel([0.293332, -1.439172, -2.525561, -0.747656, 1.570796, 1.864129],accel_mss,speed_ms,0,blend_radius_m)
      movel([0.292608, -1.438945, -2.525740, -0.747703, 1.570796, 1.863405],accel_mss,speed_ms,0,blend_radius_m)
      movel([0.291893, -1.438705, -2.525931, -0.747753, 1.570796, 1.862689],accel_mss,speed_ms,0,blend_radius_m)
      movel([0.291188, -1.438450, -2.526133, -0.747806, 1.570796, 1.861985],accel_mss,speed_ms,0,blend_radius_m)
      movel([0.290494, -1.438182, -2.526345, -0.747862, 1.570796, 1.861290],accel_mss,speed_ms,0,blend_radius_m)
      movel([0.289810, -1.437900, -2.526568, -0.747921, 1.570796, 1.860606],accel_mss,speed_ms,0,blend_radius_m)
      movel([0.289161, -1.437617, -2.526792, -0.747980, 1.570796, 1.859957],accel_mss,speed_ms,0,blend_radius_m)
      movel([0.288525, -1.437320, -2.527027, -0.748042, 1.570796, 1.859321],accel_mss,speed_ms,0,blend_radius_m)
      movel([0.287898, -1.437012, -2.527270, -0.748107, 1.570796, 1.858694],accel_mss,speed_ms,0,blend_radius_m)
      movel([0.287282, -1.436689, -2.527525, -0.748175, 1.570796, 1.858078],accel_mss,speed_ms,0,blend_radius_m)
      movel([0.286679, -1.436351, -2.527792, -0.748246, 1.570796, 1.857475],accel_mss,speed_ms,0,blend_radius_m)
      movel([0.286088, -1.436002, -2.528067, -0.748320, 1.570796, 1.856884],accel_mss,speed_ms,0,blend_radius_m)
      movel([0.285506, -1.435641, -2.528352, -0.748397, 1.570796, 1.856303],accel_mss,speed_ms,0,blend_radius_m)
      movel([0.284940, -1.435266, -2.528647, -0.748476, 1.570796, 1.855736],accel_mss,speed_ms,0,blend_radius_m)
      movel([0.284383, -1.434879, -2.528951, -0.748559, 1.570796, 1.855179],accel_mss,speed_ms,0,blend_radius_m)
      movel([0.283841, -1.434478, -2.529267, -0.748645, 1.570796, 1.854637],accel_mss,speed_ms,0,blend_radius_m)
      movel([0.283311, -1.434066, -2.529590, -0.748733, 1.570796, 1.854107],accel_mss,speed_ms,0,blend_radius_m)
      movel([0.282793, -1.433641, -2.529924, -0.748824, 1.570796, 1.853589],accel_mss,speed_ms,0,blend_radius_m)
      movel([0.282289, -1.433205, -2.530266, -0.748918, 1.570796, 1.853085],accel_mss,speed_ms,0,blend_radius_m)
      movel([0.281825, -1.432779, -2.530600, -0.749011, 1.570796, 1.852621],accel_mss,speed_ms,0,blend_radius_m)
      movel([0.281375, -1.432339, -2.530944, -0.749106, 1.570796, 1.852172],accel_mss,speed_ms,0,blend_radius_m)
      movel([0.280943, -1.431886, -2.531298, -0.749205, 1.570796, 1.851739],accel_mss,speed_ms,0,blend_radius_m)
      movel([0.280525, -1.431419, -2.531663, -0.749306, 1.570796, 1.851322],accel_mss,speed_ms,0,blend_radius_m)
      movel([0.280124, -1.430941, -2.532037, -0.749411, 1.570796, 1.850920],accel_mss,speed_ms,0,blend_radius_m)
      movel([0.279736, -1.430450, -2.532420, -0.749519, 1.570796, 1.850533],accel_mss,speed_ms,0,blend_radius_m)
      movel([0.279366, -1.429946, -2.532813, -0.749630, 1.570796, 1.850163],accel_mss,speed_ms,0,blend_radius_m)
      movel([0.279015, -1.429428, -2.533216, -0.749745, 1.570796, 1.849812],accel_mss,speed_ms,0,blend_radius_m)
      movel([0.278678, -1.428900, -2.533627, -0.749862, 1.570796, 1.849474],accel_mss,speed_ms,0,blend_radius_m)
      movel([0.278357, -1.428359, -2.534047, -0.749983, 1.570796, 1.849153],accel_mss,speed_ms,0,blend_radius_m)
      movel([0.278054, -1.427807, -2.534476, -0.750106, 1.570796, 1.848851],accel_mss,speed_ms,0,blend_radius_m)
      movel([0.277768, -1.427242, -2.534913, -0.750233, 1.570796, 1.848565],accel_mss,speed_ms,0,blend_radius_m)
      movel([0.277501, -1.426668, -2.535359, -0.750363, 1.570796, 1.848297],accel_mss,speed_ms,0,blend_radius_m)
      movel([0.277283, -1.426158, -2.535753, -0.750478, 1.570796, 1.848079],accel_mss,speed_ms,0,blend_radius_m)
      movel([0.277079, -1.425639, -2.536154, -0.750596, 1.570796, 1.847875],accel_mss,speed_ms,0,blend_radius_m)
      movel([0.276893, -1.425112, -2.536561, -0.750716, 1.570796, 1.847689],accel_mss,speed_ms,0,blend_radius_m)
      movel([0.276720, -1.424574, -2.536976, -0.750839, 1.570796, 1.847516],accel_mss,speed_ms,0,blend_radius_m)
      movel([0.276563, -1.424029, -2.537396, -0.750964, 1.570796, 1.847359],accel_mss,speed_ms,0,blend_radius_m)
      movel([0.276424, -1.423475, -2.537823, -0.751091, 1.570796, 1.847220],accel_mss,speed_ms,0,blend_radius_m)
      movel([0.276297, -1.422913, -2.538255, -0.751221, 1.570796, 1.847094],accel_mss,speed_ms,0,blend_radius_m)
      movel([0.276190, -1.422341, -2.538694, -0.751354, 1.570796, 1.846986],accel_mss,speed_ms,0,blend_radius_m)
      movel([0.276096, -1.421765, -2.539136, -0.751488, 1.570796, 1.846893],accel_mss,speed_ms,0,blend_radius_m)
      movel([0.276019, -1.421178, -2.539586, -0.751625, 1.570796, 1.846816],accel_mss,speed_ms,0,blend_radius_m)
      movel([0.275960, -1.420585, -2.540040, -0.751764, 1.570796, 1.846756],accel_mss,speed_ms,0,blend_radius_m)
      movel([0.275915, -1.419986, -2.540498, -0.751905, 1.570796, 1.846711],accel_mss,speed_ms,0,blend_radius_m)
      movel([0.275885, -1.419380, -2.540960, -0.752048, 1.570796, 1.846681],accel_mss,speed_ms,0,blend_radius_m)
      movel([0.275875, -1.418776, -2.541421, -0.752191, 1.570796, 1.846671],accel_mss,speed_ms,0,blend_radius_m)
      movel([0.275879, -1.418166, -2.541886, -0.752337, 1.570796, 1.846676],accel_mss,speed_ms,0,blend_radius_m)
      movel([0.275902, -1.417549, -2.542356, -0.752484, 1.570796, 1.846698],accel_mss,speed_ms,0,blend_radius_m)
      movel([0.275942, -1.416926, -2.542830, -0.752634, 1.570796, 1.846738],accel_mss,speed_ms,0,blend_radius_m)
      movel([0.275996, -1.416298, -2.543306, -0.752785, 1.570796, 1.846792],accel_mss,speed_ms,0,blend_radius_m)
      movel([0.276069, -1.415665, -2.543786, -0.752938, 1.570796, 1.846866],accel_mss,speed_ms,0,blend_radius_m)
      movel([0.276161, -1.415026, -2.544270, -0.753093, 1.570796, 1.846957],accel_mss,speed_ms,0,blend_radius_m)
      movel([0.276266, -1.414385, -2.544755, -0.753249, 1.570796, 1.847062],accel_mss,speed_ms,0,blend_radius_m)
      movel([0.276391, -1.413736, -2.545244, -0.753408, 1.570796, 1.847188],accel_mss,speed_ms,0,blend_radius_m)
      movel([0.276531, -1.413086, -2.545735, -0.753568, 1.570796, 1.847327],accel_mss,speed_ms,0,blend_radius_m)
      movel([0.276689, -1.412433, -2.546227, -0.753729, 1.570796, 1.847485],accel_mss,speed_ms,0,blend_radius_m)
      movel([0.276862, -1.411775, -2.546722, -0.753892, 1.570796, 1.847658],accel_mss,speed_ms,0,blend_radius_m)
      movel([0.277054, -1.411115, -2.547218, -0.754056, 1.570796, 1.847850],accel_mss,speed_ms,0,blend_radius_m)
      movel([0.277260, -1.410452, -2.547716, -0.754221, 1.570796, 1.848056],accel_mss,speed_ms,0,blend_radius_m)
      movel([0.277485, -1.409789, -2.548213, -0.754387, 1.570796, 1.848281],accel_mss,speed_ms,0,blend_radius_m)
      movel([0.277723, -1.409123, -2.548711, -0.754555, 1.570796, 1.848520],accel_mss,speed_ms,0,blend_radius_m)
      movel([0.277980, -1.408457, -2.549209, -0.754723, 1.570796, 1.848777],accel_mss,speed_ms,0,blend_radius_m)
      movel([0.278254, -1.407789, -2.549708, -0.754892, 1.570796, 1.849051],accel_mss,speed_ms,0,blend_radius_m)
      movel([0.278542, -1.407120, -2.550207, -0.755063, 1.570796, 1.849338],accel_mss,speed_ms,0,blend_radius_m)
      movel([0.278849, -1.406448, -2.550707, -0.755234, 1.570796, 1.849645],accel_mss,speed_ms,0,blend_radius_m)
      movel([0.279169, -1.405779, -2.551205, -0.755406, 1.570796, 1.849965],accel_mss,speed_ms,0,blend_radius_m)
      movel([0.279507, -1.405108, -2.551702, -0.755578, 1.570796, 1.850303],accel_mss,speed_ms,0,blend_radius_m)
      movel([0.279859, -1.404440, -2.552198, -0.755751, 1.570796, 1.850655],accel_mss,speed_ms,0,blend_radius_m)
      movel([0.280229, -1.403771, -2.552693, -0.755924, 1.570796, 1.851025],accel_mss,speed_ms,0,blend_radius_m)
      movel([0.280613, -1.403104, -2.553186, -0.756098, 1.570796, 1.851409],accel_mss,speed_ms,0,blend_radius_m)
      movel([0.281010, -1.402438, -2.553679, -0.756272, 1.570796, 1.851806],accel_mss,speed_ms,0,blend_radius_m)
      movel([0.281429, -1.401768, -2.554173, -0.756448, 1.570796, 1.852226],accel_mss,speed_ms,0,blend_radius_m)
      movel([0.281862, -1.401100, -2.554665, -0.756624, 1.570796, 1.852658],accel_mss,speed_ms,0,blend_radius_m)
      movel([0.282308, -1.400434, -2.555155, -0.756800, 1.570796, 1.853104],accel_mss,speed_ms,0,blend_radius_m)
      movel([0.282769, -1.399770, -2.555643, -0.756976, 1.570796, 1.853566],accel_mss,speed_ms,0,blend_radius_m)
      movel([0.283243, -1.399113, -2.556125, -0.757151, 1.570796, 1.854039],accel_mss,speed_ms,0,blend_radius_m)
      movel([0.283733, -1.398455, -2.556607, -0.757327, 1.570796, 1.854530],accel_mss,speed_ms,0,blend_radius_m)
      movel([0.284236, -1.397804, -2.557084, -0.757501, 1.570796, 1.855032],accel_mss,speed_ms,0,blend_radius_m)
      movel([0.284751, -1.397157, -2.557557, -0.757675, 1.570796, 1.855547],accel_mss,speed_ms,0,blend_radius_m)
      movel([0.285279, -1.396512, -2.558027, -0.757850, 1.570796, 1.856075],accel_mss,speed_ms,0,blend_radius_m)
      movel([0.285822, -1.395874, -2.558493, -0.758022, 1.570796, 1.856618],accel_mss,speed_ms,0,blend_radius_m)
      movel([0.286375, -1.395243, -2.558952, -0.758194, 1.570796, 1.857171],accel_mss,speed_ms,0,blend_radius_m)
      movel([0.286940, -1.394616, -2.559408, -0.758365, 1.570796, 1.857737],accel_mss,speed_ms,0,blend_radius_m)
      movel([0.287521, -1.393993, -2.559860, -0.758536, 1.570796, 1.858317],accel_mss,speed_ms,0,blend_radius_m)
      movel([0.288191, -1.393294, -2.560367, -0.758728, 1.570796, 1.858987],accel_mss,speed_ms,0,blend_radius_m)
      movel([0.288872, -1.392604, -2.560867, -0.758918, 1.570796, 1.859668],accel_mss,speed_ms,0,blend_radius_m)
      movel([0.289568, -1.391920, -2.561362, -0.759107, 1.570796, 1.860364],accel_mss,speed_ms,0,blend_radius_m)
      movel([0.290276, -1.391243, -2.561851, -0.759295, 1.570796, 1.861072],accel_mss,speed_ms,0,blend_radius_m)
      movel([0.290993, -1.390575, -2.562333, -0.759481, 1.570796, 1.861790],accel_mss,speed_ms,0,blend_radius_m)
      movel([0.291723, -1.389914, -2.562809, -0.759666, 1.570796, 1.862520],accel_mss,speed_ms,0,blend_radius_m)
      movel([0.292464, -1.389265, -2.563276, -0.759848, 1.570796, 1.863260],accel_mss,speed_ms,0,blend_radius_m)
      movel([0.293216, -1.388624, -2.563736, -0.760028, 1.570796, 1.864013],accel_mss,speed_ms,0,blend_radius_m)
      movel([0.293979, -1.387991, -2.564191, -0.760207, 1.570796, 1.864775],accel_mss,speed_ms,0,blend_radius_m)
      movel([0.294749, -1.387369, -2.564636, -0.760383, 1.570796, 1.865546],accel_mss,speed_ms,0,blend_radius_m)
      movel([0.295532, -1.386757, -2.565075, -0.760557, 1.570796, 1.866328],accel_mss,speed_ms,0,blend_radius_m)
      movel([0.296344, -1.386139, -2.565516, -0.760734, 1.570796, 1.867141],accel_mss,speed_ms,0,blend_radius_m)
      movel([0.297164, -1.385531, -2.565951, -0.760908, 1.570796, 1.867960],accel_mss,speed_ms,0,blend_radius_m)
      movel([0.297994, -1.384932, -2.566378, -0.761079, 1.570796, 1.868791],accel_mss,speed_ms,0,blend_radius_m)
      movel([0.298832, -1.384343, -2.566797, -0.761249, 1.570796, 1.869629],accel_mss,speed_ms,0,blend_radius_m)
      movel([0.299675, -1.383769, -2.567205, -0.761414, 1.570796, 1.870471],accel_mss,speed_ms,0,blend_radius_m)
      movel([0.300528, -1.383203, -2.567608, -0.761578, 1.570796, 1.871324],accel_mss,speed_ms,0,blend_radius_m)
      movel([0.301384, -1.382651, -2.568000, -0.761738, 1.570796, 1.872180],accel_mss,speed_ms,0,blend_radius_m)
      movel([0.302251, -1.382109, -2.568384, -0.761896, 1.570796, 1.873047],accel_mss,speed_ms,0,blend_radius_m)
      movel([0.303121, -1.381579, -2.568759, -0.762051, 1.570796, 1.873918],accel_mss,speed_ms,0,blend_radius_m)
      movel([0.303995, -1.381063, -2.569125, -0.762202, 1.570796, 1.874792],accel_mss,speed_ms,0,blend_radius_m)
      movel([0.304877, -1.380558, -2.569481, -0.762350, 1.570796, 1.875674],accel_mss,speed_ms,0,blend_radius_m)
      movel([0.305803, -1.380045, -2.569843, -0.762500, 1.570796, 1.876599],accel_mss,speed_ms,0,blend_radius_m)
      movel([0.306731, -1.379545, -2.570196, -0.762648, 1.570796, 1.877527],accel_mss,speed_ms,0,blend_radius_m)
      movel([0.307665, -1.379058, -2.570539, -0.762792, 1.570796, 1.878462],accel_mss,speed_ms,0,blend_radius_m)
      movel([0.308600, -1.378586, -2.570871, -0.762931, 1.570796, 1.879396],accel_mss,speed_ms,0,blend_radius_m)
      movel([0.309540, -1.378128, -2.571194, -0.763067, 1.570796, 1.880336],accel_mss,speed_ms,0,blend_radius_m)
      movel([0.310486, -1.377682, -2.571507, -0.763200, 1.570796, 1.881282],accel_mss,speed_ms,0,blend_radius_m)
      movel([0.311432, -1.377249, -2.571811, -0.763329, 1.570796, 1.882229],accel_mss,speed_ms,0,blend_radius_m)
      movel([0.312381, -1.376832, -2.572104, -0.763453, 1.570796, 1.883178],accel_mss,speed_ms,0,blend_radius_m)
      movel([0.313330, -1.376431, -2.572385, -0.763574, 1.570796, 1.884126],accel_mss,speed_ms,0,blend_radius_m)
      movel([0.314282, -1.376043, -2.572657, -0.763690, 1.570796, 1.885078],accel_mss,speed_ms,0,blend_radius_m)
      movel([0.315236, -1.375670, -2.572917, -0.763802, 1.570796, 1.886032],accel_mss,speed_ms,0,blend_radius_m)
      movel([0.316337, -1.375256, -2.573207, -0.763926, 1.570796, 1.887134],accel_mss,speed_ms,0,blend_radius_m)
      movel([0.317438, -1.374860, -2.573483, -0.764046, 1.570796, 1.888234],accel_mss,speed_ms,0,blend_radius_m)
      movel([0.318538, -1.374480, -2.573749, -0.764160, 1.570796, 1.889335],accel_mss,speed_ms,0,blend_radius_m)
      movel([0.319640, -1.374118, -2.574001, -0.764270, 1.570796, 1.890436],accel_mss,speed_ms,0,blend_radius_m)
      movel([0.320741, -1.373773, -2.574242, -0.764375, 1.570796, 1.891538],accel_mss,speed_ms,0,blend_radius_m)
      movel([0.321839, -1.373446, -2.574469, -0.764474, 1.570796, 1.892635],accel_mss,speed_ms,0,blend_radius_m)
      movel([0.322939, -1.373136, -2.574685, -0.764568, 1.570796, 1.893735],accel_mss,speed_ms,0,blend_radius_m)
      movel([0.324035, -1.372844, -2.574888, -0.764657, 1.570796, 1.894831],accel_mss,speed_ms,0,blend_radius_m)
      movel([0.325127, -1.372572, -2.575078, -0.764740, 1.570796, 1.895923],accel_mss,speed_ms,0,blend_radius_m)
      movel([0.326218, -1.372315, -2.575256, -0.764818, 1.570796, 1.897014],accel_mss,speed_ms,0,blend_radius_m)
      movel([0.327079, -1.372126, -2.575387, -0.764876, 1.570796, 1.897875],accel_mss,speed_ms,0,blend_radius_m)
      movel([0.327938, -1.371949, -2.575510, -0.764930, 1.570796, 1.898734],accel_mss,speed_ms,0,blend_radius_m)
      movel([0.328792, -1.371786, -2.575623, -0.764980, 1.570796, 1.899588],accel_mss,speed_ms,0,blend_radius_m)
      movel([0.329644, -1.371635, -2.575728, -0.765026, 1.570796, 1.900441],accel_mss,speed_ms,0,blend_radius_m)
      movel([0.330936, -1.371424, -2.575874, -0.765091, 1.570796, 1.901732],accel_mss,speed_ms,0,blend_radius_m)
      movel([0.332225, -1.371233, -2.576007, -0.765149, 1.570796, 1.903021],accel_mss,speed_ms,0,blend_radius_m)
      movel([0.333506, -1.371057, -2.576129, -0.765204, 1.570796, 1.904303],accel_mss,speed_ms,0,blend_radius_m)
      movel([0.334686, -1.370912, -2.576229, -0.765248, 1.570796, 1.905482],accel_mss,speed_ms,0,blend_radius_m)
      movel([0.335859, -1.370778, -2.576322, -0.765289, 1.570796, 1.906656],accel_mss,speed_ms,0,blend_radius_m)
      movel([0.337030, -1.370659, -2.576404, -0.765326, 1.570796, 1.907827],accel_mss,speed_ms,0,blend_radius_m)
      movel([0.337336, -1.370638, -2.576419, -0.765332, 1.570796, 1.908132],accel_mss,speed_ms,0,blend_radius_m)
      movel([0.337636, -1.370633, -2.576422, -0.765334, 1.570796, 1.908432],accel_mss,speed_ms,0,blend_radius_m)
      movel([0.337928, -1.370645, -2.576414, -0.765330, 1.570796, 1.908724],accel_mss,speed_ms,0,blend_radius_m)
      movel([0.338213, -1.370673, -2.576395, -0.765322, 1.570796, 1.909010],accel_mss,speed_ms,0,blend_radius_m)
      movel([0.338485, -1.370719, -2.576362, -0.765307, 1.570796, 1.909281],accel_mss,speed_ms,0,blend_radius_m)
      speed_ms = 0.003
      movel([0.338485, -1.374028, -2.577865, -0.760496, 1.570796, 1.909281],accel_mss,speed_ms,0,blend_radius_m)
      speed_ms = 0.007
      movel([0.338879, -1.374108, -2.577810, -0.760472, 1.570796, 1.909676],accel_mss,speed_ms,0,blend_radius_m)
      movel([0.326050, -1.409128, -2.552548, -0.750713, 1.570796, 1.896846],accel_mss,speed_ms,0,blend_radius_m)
      movel([0.321364, -1.422111, -2.542725, -0.747554, 1.570796, 1.892160],accel_mss,speed_ms,0,blend_radius_m)
      movel([0.317469, -1.432959, -2.534322, -0.745108, 1.570796, 1.888265],accel_mss,speed_ms,0,blend_radius_m)
      movel([0.314074, -1.442467, -2.526812, -0.743110, 1.570796, 1.884870],accel_mss,speed_ms,0,blend_radius_m)
      movel([0.313964, -1.442750, -2.526586, -0.743053, 1.570796, 1.884760],accel_mss,speed_ms,0,blend_radius_m)
      movel([0.313839, -1.443032, -2.526361, -0.742996, 1.570796, 1.884635],accel_mss,speed_ms,0,blend_radius_m)
      movel([0.313503, -1.443738, -2.525797, -0.742854, 1.570796, 1.884299],accel_mss,speed_ms,0,blend_radius_m)
      movel([0.310537, -1.443941, -2.525635, -0.742813, 1.570796, 1.881334],accel_mss,speed_ms,0,blend_radius_m)
      movel([0.309649, -1.443998, -2.525590, -0.742802, 1.570796, 1.880445],accel_mss,speed_ms,0,blend_radius_m)
      movel([0.308768, -1.444038, -2.525557, -0.742794, 1.570796, 1.879564],accel_mss,speed_ms,0,blend_radius_m)
      movel([0.307891, -1.444067, -2.525534, -0.742788, 1.570796, 1.878688],accel_mss,speed_ms,0,blend_radius_m)
      movel([0.307019, -1.444082, -2.525522, -0.742785, 1.570796, 1.877816],accel_mss,speed_ms,0,blend_radius_m)
      movel([0.306154, -1.444084, -2.525521, -0.742784, 1.570796, 1.876950],accel_mss,speed_ms,0,blend_radius_m)
      movel([0.305293, -1.444073, -2.525529, -0.742787, 1.570796, 1.876089],accel_mss,speed_ms,0,blend_radius_m)
      movel([0.304439, -1.444047, -2.525550, -0.742792, 1.570796, 1.875235],accel_mss,speed_ms,0,blend_radius_m)
      movel([0.303591, -1.444009, -2.525580, -0.742799, 1.570796, 1.874388],accel_mss,speed_ms,0,blend_radius_m)
      movel([0.302750, -1.443957, -2.525622, -0.742810, 1.570796, 1.873547],accel_mss,speed_ms,0,blend_radius_m)
      movel([0.301914, -1.443892, -2.525674, -0.742823, 1.570796, 1.872710],accel_mss,speed_ms,0,blend_radius_m)
      movel([0.301086, -1.443812, -2.525738, -0.742839, 1.570796, 1.871882],accel_mss,speed_ms,0,blend_radius_m)
      movel([0.300266, -1.443721, -2.525811, -0.742857, 1.570796, 1.871063],accel_mss,speed_ms,0,blend_radius_m)
      movel([0.299452, -1.443614, -2.525897, -0.742879, 1.570796, 1.870248],accel_mss,speed_ms,0,blend_radius_m)
      movel([0.298658, -1.443497, -2.525989, -0.742902, 1.570796, 1.869454],accel_mss,speed_ms,0,blend_radius_m)
      movel([0.297871, -1.443365, -2.526095, -0.742929, 1.570796, 1.868667],accel_mss,speed_ms,0,blend_radius_m)
      movel([0.297094, -1.443221, -2.526210, -0.742958, 1.570796, 1.867890],accel_mss,speed_ms,0,blend_radius_m)
      movel([0.296324, -1.443060, -2.526339, -0.742990, 1.570796, 1.867120],accel_mss,speed_ms,0,blend_radius_m)
      movel([0.295562, -1.442888, -2.526476, -0.743025, 1.570796, 1.866359],accel_mss,speed_ms,0,blend_radius_m)
      movel([0.294809, -1.442703, -2.526624, -0.743063, 1.570796, 1.865605],accel_mss,speed_ms,0,blend_radius_m)
      movel([0.294067, -1.442502, -2.526784, -0.743103, 1.570796, 1.864863],accel_mss,speed_ms,0,blend_radius_m)
      movel([0.293332, -1.442289, -2.526954, -0.743147, 1.570796, 1.864129],accel_mss,speed_ms,0,blend_radius_m)
      movel([0.292608, -1.442063, -2.527134, -0.743192, 1.570796, 1.863405],accel_mss,speed_ms,0,blend_radius_m)
      movel([0.291893, -1.441823, -2.527325, -0.743241, 1.570796, 1.862689],accel_mss,speed_ms,0,blend_radius_m)
      movel([0.291188, -1.441569, -2.527527, -0.743293, 1.570796, 1.861985],accel_mss,speed_ms,0,blend_radius_m)
      movel([0.290494, -1.441302, -2.527739, -0.743348, 1.570796, 1.861290],accel_mss,speed_ms,0,blend_radius_m)
      movel([0.289810, -1.441021, -2.527963, -0.743405, 1.570796, 1.860606],accel_mss,speed_ms,0,blend_radius_m)
      movel([0.289161, -1.440739, -2.528187, -0.743463, 1.570796, 1.859957],accel_mss,speed_ms,0,blend_radius_m)
      movel([0.288525, -1.440442, -2.528423, -0.743524, 1.570796, 1.859321],accel_mss,speed_ms,0,blend_radius_m)
      movel([0.287898, -1.440135, -2.528667, -0.743588, 1.570796, 1.858694],accel_mss,speed_ms,0,blend_radius_m)
      movel([0.287282, -1.439813, -2.528922, -0.743654, 1.570796, 1.858078],accel_mss,speed_ms,0,blend_radius_m)
      movel([0.286679, -1.439476, -2.529189, -0.743724, 1.570796, 1.857475],accel_mss,speed_ms,0,blend_radius_m)
      movel([0.286088, -1.439128, -2.529465, -0.743796, 1.570796, 1.856884],accel_mss,speed_ms,0,blend_radius_m)
      movel([0.285506, -1.438768, -2.529750, -0.743871, 1.570796, 1.856303],accel_mss,speed_ms,0,blend_radius_m)
      movel([0.284940, -1.438394, -2.530046, -0.743949, 1.570796, 1.855736],accel_mss,speed_ms,0,blend_radius_m)
      movel([0.284383, -1.438008, -2.530351, -0.744030, 1.570796, 1.855179],accel_mss,speed_ms,0,blend_radius_m)
      movel([0.283841, -1.437609, -2.530667, -0.744114, 1.570796, 1.854637],accel_mss,speed_ms,0,blend_radius_m)
      movel([0.283311, -1.437198, -2.530991, -0.744200, 1.570796, 1.854107],accel_mss,speed_ms,0,blend_radius_m)
      movel([0.282793, -1.436774, -2.531325, -0.744290, 1.570796, 1.853589],accel_mss,speed_ms,0,blend_radius_m)
      movel([0.282289, -1.436339, -2.531668, -0.744382, 1.570796, 1.853085],accel_mss,speed_ms,0,blend_radius_m)
      movel([0.281825, -1.435915, -2.532002, -0.744472, 1.570796, 1.852621],accel_mss,speed_ms,0,blend_radius_m)
      movel([0.281375, -1.435476, -2.532347, -0.744565, 1.570796, 1.852172],accel_mss,speed_ms,0,blend_radius_m)
      movel([0.280943, -1.435024, -2.532703, -0.744662, 1.570796, 1.851739],accel_mss,speed_ms,0,blend_radius_m)
      movel([0.280525, -1.434559, -2.533068, -0.744762, 1.570796, 1.851322],accel_mss,speed_ms,0,blend_radius_m)
      movel([0.280124, -1.434082, -2.533443, -0.744865, 1.570796, 1.850920],accel_mss,speed_ms,0,blend_radius_m)
      movel([0.279736, -1.433593, -2.533826, -0.744970, 1.570796, 1.850533],accel_mss,speed_ms,0,blend_radius_m)
      movel([0.279366, -1.433090, -2.534220, -0.745079, 1.570796, 1.850163],accel_mss,speed_ms,0,blend_radius_m)
      movel([0.279015, -1.432573, -2.534624, -0.745192, 1.570796, 1.849812],accel_mss,speed_ms,0,blend_radius_m)
      movel([0.278678, -1.432046, -2.535036, -0.745306, 1.570796, 1.849474],accel_mss,speed_ms,0,blend_radius_m)
      movel([0.278357, -1.431508, -2.535457, -0.745424, 1.570796, 1.849153],accel_mss,speed_ms,0,blend_radius_m)
      movel([0.278054, -1.430957, -2.535886, -0.745546, 1.570796, 1.848851],accel_mss,speed_ms,0,blend_radius_m)
      movel([0.277768, -1.430394, -2.536325, -0.745670, 1.570796, 1.848565],accel_mss,speed_ms,0,blend_radius_m)
      movel([0.277501, -1.429821, -2.536771, -0.745797, 1.570796, 1.848297],accel_mss,speed_ms,0,blend_radius_m)
      movel([0.277283, -1.429313, -2.537166, -0.745910, 1.570796, 1.848079],accel_mss,speed_ms,0,blend_radius_m)
      movel([0.277079, -1.428795, -2.537568, -0.746025, 1.570796, 1.847875],accel_mss,speed_ms,0,blend_radius_m)
      movel([0.276893, -1.428269, -2.537976, -0.746143, 1.570796, 1.847689],accel_mss,speed_ms,0,blend_radius_m)
      movel([0.276720, -1.427734, -2.538392, -0.746264, 1.570796, 1.847516],accel_mss,speed_ms,0,blend_radius_m)
      movel([0.276563, -1.427190, -2.538813, -0.746386, 1.570796, 1.847359],accel_mss,speed_ms,0,blend_radius_m)
      movel([0.276424, -1.426638, -2.539240, -0.746511, 1.570796, 1.847220],accel_mss,speed_ms,0,blend_radius_m)
      movel([0.276297, -1.426077, -2.539673, -0.746639, 1.570796, 1.847094],accel_mss,speed_ms,0,blend_radius_m)
      movel([0.276190, -1.425507, -2.540113, -0.746769, 1.570796, 1.846986],accel_mss,speed_ms,0,blend_radius_m)
      movel([0.276096, -1.424932, -2.540557, -0.746900, 1.570796, 1.846893],accel_mss,speed_ms,0,blend_radius_m)
      movel([0.276019, -1.424347, -2.541007, -0.747035, 1.570796, 1.846816],accel_mss,speed_ms,0,blend_radius_m)
      movel([0.275960, -1.423756, -2.541462, -0.747171, 1.570796, 1.846756],accel_mss,speed_ms,0,blend_radius_m)
      movel([0.275915, -1.423158, -2.541921, -0.747310, 1.570796, 1.846711],accel_mss,speed_ms,0,blend_radius_m)
      movel([0.275885, -1.422554, -2.542385, -0.747450, 1.570796, 1.846681],accel_mss,speed_ms,0,blend_radius_m)
      movel([0.275875, -1.421952, -2.542846, -0.747591, 1.570796, 1.846671],accel_mss,speed_ms,0,blend_radius_m)
      movel([0.275879, -1.421343, -2.543312, -0.747733, 1.570796, 1.846676],accel_mss,speed_ms,0,blend_radius_m)
      movel([0.275902, -1.420728, -2.543783, -0.747878, 1.570796, 1.846698],accel_mss,speed_ms,0,blend_radius_m)
      movel([0.275942, -1.420107, -2.544258, -0.748025, 1.570796, 1.846738],accel_mss,speed_ms,0,blend_radius_m)
      movel([0.275996, -1.419481, -2.544735, -0.748173, 1.570796, 1.846792],accel_mss,speed_ms,0,blend_radius_m)
      movel([0.276069, -1.418850, -2.545216, -0.748323, 1.570796, 1.846866],accel_mss,speed_ms,0,blend_radius_m)
      movel([0.276161, -1.418213, -2.545701, -0.748476, 1.570796, 1.846957],accel_mss,speed_ms,0,blend_radius_m)
      movel([0.276266, -1.417573, -2.546187, -0.748629, 1.570796, 1.847062],accel_mss,speed_ms,0,blend_radius_m)
      movel([0.276391, -1.416927, -2.546677, -0.748785, 1.570796, 1.847188],accel_mss,speed_ms,0,blend_radius_m)
      movel([0.276531, -1.416278, -2.547169, -0.748942, 1.570796, 1.847327],accel_mss,speed_ms,0,blend_radius_m)
      movel([0.276689, -1.415627, -2.547662, -0.749100, 1.570796, 1.847485],accel_mss,speed_ms,0,blend_radius_m)
      movel([0.276862, -1.414971, -2.548158, -0.749260, 1.570796, 1.847658],accel_mss,speed_ms,0,blend_radius_m)
      movel([0.277054, -1.414312, -2.548656, -0.749421, 1.570796, 1.847850],accel_mss,speed_ms,0,blend_radius_m)
      movel([0.277260, -1.413652, -2.549154, -0.749583, 1.570796, 1.848056],accel_mss,speed_ms,0,blend_radius_m)
      movel([0.277485, -1.412990, -2.549652, -0.749747, 1.570796, 1.848281],accel_mss,speed_ms,0,blend_radius_m)
      movel([0.277723, -1.412327, -2.550151, -0.749911, 1.570796, 1.848520],accel_mss,speed_ms,0,blend_radius_m)
      movel([0.277980, -1.411662, -2.550650, -0.750076, 1.570796, 1.848777],accel_mss,speed_ms,0,blend_radius_m)
      movel([0.278254, -1.410996, -2.551151, -0.750243, 1.570796, 1.849051],accel_mss,speed_ms,0,blend_radius_m)
      movel([0.278542, -1.410329, -2.551650, -0.750410, 1.570796, 1.849338],accel_mss,speed_ms,0,blend_radius_m)
      movel([0.278849, -1.409659, -2.552151, -0.750579, 1.570796, 1.849645],accel_mss,speed_ms,0,blend_radius_m)
      movel([0.279169, -1.408991, -2.552650, -0.750747, 1.570796, 1.849965],accel_mss,speed_ms,0,blend_radius_m)
      movel([0.279507, -1.408323, -2.553149, -0.750917, 1.570796, 1.850303],accel_mss,speed_ms,0,blend_radius_m)
      movel([0.279859, -1.407656, -2.553646, -0.751087, 1.570796, 1.850655],accel_mss,speed_ms,0,blend_radius_m)
      movel([0.280229, -1.406989, -2.554142, -0.751257, 1.570796, 1.851025],accel_mss,speed_ms,0,blend_radius_m)
      movel([0.280613, -1.406325, -2.554637, -0.751428, 1.570796, 1.851409],accel_mss,speed_ms,0,blend_radius_m)
      movel([0.281010, -1.405659, -2.555130, -0.751599, 1.570796, 1.851806],accel_mss,speed_ms,0,blend_radius_m)
      movel([0.281429, -1.404991, -2.555626, -0.751772, 1.570796, 1.852226],accel_mss,speed_ms,0,blend_radius_m)
      movel([0.281862, -1.404325, -2.556119, -0.751945, 1.570796, 1.852658],accel_mss,speed_ms,0,blend_radius_m)
      movel([0.282308, -1.403661, -2.556610, -0.752118, 1.570796, 1.853104],accel_mss,speed_ms,0,blend_radius_m)
      movel([0.282769, -1.402999, -2.557098, -0.752291, 1.570796, 1.853566],accel_mss,speed_ms,0,blend_radius_m)
      movel([0.283243, -1.402344, -2.557582, -0.752463, 1.570796, 1.854039],accel_mss,speed_ms,0,blend_radius_m)
      movel([0.283733, -1.401688, -2.558065, -0.752636, 1.570796, 1.854530],accel_mss,speed_ms,0,blend_radius_m)
      movel([0.284236, -1.401038, -2.558543, -0.752808, 1.570796, 1.855032],accel_mss,speed_ms,0,blend_radius_m)
      movel([0.284751, -1.400393, -2.559017, -0.752979, 1.570796, 1.855547],accel_mss,speed_ms,0,blend_radius_m)
      movel([0.285279, -1.399751, -2.559488, -0.753150, 1.570796, 1.856075],accel_mss,speed_ms,0,blend_radius_m)
      movel([0.285822, -1.399114, -2.559954, -0.753320, 1.570796, 1.856618],accel_mss,speed_ms,0,blend_radius_m)
      movel([0.286375, -1.398484, -2.560415, -0.753489, 1.570796, 1.857171],accel_mss,speed_ms,0,blend_radius_m)
      movel([0.286940, -1.397859, -2.560872, -0.753658, 1.570796, 1.857737],accel_mss,speed_ms,0,blend_radius_m)
      movel([0.287521, -1.397238, -2.561325, -0.753825, 1.570796, 1.858317],accel_mss,speed_ms,0,blend_radius_m)
      movel([0.288191, -1.396541, -2.561833, -0.754014, 1.570796, 1.858987],accel_mss,speed_ms,0,blend_radius_m)
      movel([0.288872, -1.395853, -2.562334, -0.754201, 1.570796, 1.859668],accel_mss,speed_ms,0,blend_radius_m)
      movel([0.289568, -1.395171, -2.562830, -0.754388, 1.570796, 1.860364],accel_mss,speed_ms,0,blend_radius_m)
      movel([0.290276, -1.394496, -2.563320, -0.754573, 1.570796, 1.861072],accel_mss,speed_ms,0,blend_radius_m)
      movel([0.290993, -1.393830, -2.563803, -0.754756, 1.570796, 1.861790],accel_mss,speed_ms,0,blend_radius_m)
      movel([0.291723, -1.393171, -2.564280, -0.754938, 1.570796, 1.862520],accel_mss,speed_ms,0,blend_radius_m)
      movel([0.292464, -1.392523, -2.564749, -0.755117, 1.570796, 1.863260],accel_mss,speed_ms,0,blend_radius_m)
      movel([0.293216, -1.391884, -2.565210, -0.755295, 1.570796, 1.864013],accel_mss,speed_ms,0,blend_radius_m)
      movel([0.293979, -1.391253, -2.565665, -0.755471, 1.570796, 1.864775],accel_mss,speed_ms,0,blend_radius_m)
      movel([0.294749, -1.390633, -2.566112, -0.755644, 1.570796, 1.865546],accel_mss,speed_ms,0,blend_radius_m)
      movel([0.295532, -1.390022, -2.566551, -0.755816, 1.570796, 1.866328],accel_mss,speed_ms,0,blend_radius_m)
      movel([0.296344, -1.389406, -2.566994, -0.755989, 1.570796, 1.867141],accel_mss,speed_ms,0,blend_radius_m)
      movel([0.297164, -1.388799, -2.567429, -0.756160, 1.570796, 1.867960],accel_mss,speed_ms,0,blend_radius_m)
      movel([0.297994, -1.388202, -2.567857, -0.756329, 1.570796, 1.868791],accel_mss,speed_ms,0,blend_radius_m)
      movel([0.298832, -1.387615, -2.568277, -0.756496, 1.570796, 1.869629],accel_mss,speed_ms,0,blend_radius_m)
      movel([0.299675, -1.387043, -2.568687, -0.756659, 1.570796, 1.870471],accel_mss,speed_ms,0,blend_radius_m)
      movel([0.300528, -1.386477, -2.569091, -0.756821, 1.570796, 1.871324],accel_mss,speed_ms,0,blend_radius_m)
      movel([0.301384, -1.385927, -2.569483, -0.756979, 1.570796, 1.872180],accel_mss,speed_ms,0,blend_radius_m)
      movel([0.302251, -1.385387, -2.569868, -0.757134, 1.570796, 1.873047],accel_mss,speed_ms,0,blend_radius_m)
      movel([0.303121, -1.384859, -2.570244, -0.757286, 1.570796, 1.873918],accel_mss,speed_ms,0,blend_radius_m)
      movel([0.303995, -1.384343, -2.570611, -0.757435, 1.570796, 1.874792],accel_mss,speed_ms,0,blend_radius_m)
      movel([0.304877, -1.383840, -2.570968, -0.757581, 1.570796, 1.875674],accel_mss,speed_ms,0,blend_radius_m)
      movel([0.305803, -1.383329, -2.571331, -0.757729, 1.570796, 1.876599],accel_mss,speed_ms,0,blend_radius_m)
      movel([0.306731, -1.382830, -2.571684, -0.757874, 1.570796, 1.877527],accel_mss,speed_ms,0,blend_radius_m)
      movel([0.307665, -1.382344, -2.572028, -0.758016, 1.570796, 1.878462],accel_mss,speed_ms,0,blend_radius_m)
      movel([0.308600, -1.381874, -2.572361, -0.758154, 1.570796, 1.879396],accel_mss,speed_ms,0,blend_radius_m)
      movel([0.309540, -1.381416, -2.572685, -0.758288, 1.570796, 1.880336],accel_mss,speed_ms,0,blend_radius_m)
      movel([0.310486, -1.380971, -2.572999, -0.758419, 1.570796, 1.881282],accel_mss,speed_ms,0,blend_radius_m)
      movel([0.311432, -1.380540, -2.573303, -0.758546, 1.570796, 1.882229],accel_mss,speed_ms,0,blend_radius_m)
      movel([0.312381, -1.380124, -2.573596, -0.758669, 1.570796, 1.883178],accel_mss,speed_ms,0,blend_radius_m)
      movel([0.313330, -1.379724, -2.573878, -0.758787, 1.570796, 1.884126],accel_mss,speed_ms,0,blend_radius_m)
      movel([0.314282, -1.379337, -2.574151, -0.758902, 1.570796, 1.885078],accel_mss,speed_ms,0,blend_radius_m)
      movel([0.315236, -1.378965, -2.574412, -0.759012, 1.570796, 1.886032],accel_mss,speed_ms,0,blend_radius_m)
      movel([0.316337, -1.378552, -2.574702, -0.759135, 1.570796, 1.887134],accel_mss,speed_ms,0,blend_radius_m)
      movel([0.317438, -1.378157, -2.574980, -0.759252, 1.570796, 1.888234],accel_mss,speed_ms,0,blend_radius_m)
      movel([0.318538, -1.377778, -2.575245, -0.759365, 1.570796, 1.889335],accel_mss,speed_ms,0,blend_radius_m)
      movel([0.319640, -1.377418, -2.575498, -0.759473, 1.570796, 1.890436],accel_mss,speed_ms,0,blend_radius_m)
      movel([0.320741, -1.377073, -2.575739, -0.759576, 1.570796, 1.891538],accel_mss,speed_ms,0,blend_radius_m)
      movel([0.321839, -1.376747, -2.575967, -0.759674, 1.570796, 1.892635],accel_mss,speed_ms,0,blend_radius_m)
      movel([0.322939, -1.376438, -2.576184, -0.759767, 1.570796, 1.893735],accel_mss,speed_ms,0,blend_radius_m)
      movel([0.324035, -1.376147, -2.576387, -0.759855, 1.570796, 1.894831],accel_mss,speed_ms,0,blend_radius_m)
      movel([0.325127, -1.375875, -2.576577, -0.759937, 1.570796, 1.895923],accel_mss,speed_ms,0,blend_radius_m)
      movel([0.326218, -1.375620, -2.576756, -0.760014, 1.570796, 1.897014],accel_mss,speed_ms,0,blend_radius_m)
      movel([0.327079, -1.375431, -2.576887, -0.760071, 1.570796, 1.897875],accel_mss,speed_ms,0,blend_radius_m)
      movel([0.327938, -1.375254, -2.577011, -0.760124, 1.570796, 1.898734],accel_mss,speed_ms,0,blend_radius_m)
      movel([0.328792, -1.375092, -2.577124, -0.760173, 1.570796, 1.899588],accel_mss,speed_ms,0,blend_radius_m)
      movel([0.329644, -1.374941, -2.577229, -0.760219, 1.570796, 1.900441],accel_mss,speed_ms,0,blend_radius_m)
      movel([0.330936, -1.374731, -2.577376, -0.760282, 1.570796, 1.901732],accel_mss,speed_ms,0,blend_radius_m)
      movel([0.332225, -1.374540, -2.577509, -0.760340, 1.570796, 1.903021],accel_mss,speed_ms,0,blend_radius_m)
      movel([0.333506, -1.374364, -2.577631, -0.760394, 1.570796, 1.904303],accel_mss,speed_ms,0,blend_radius_m)
      movel([0.334686, -1.374220, -2.577731, -0.760437, 1.570796, 1.905482],accel_mss,speed_ms,0,blend_radius_m)
      movel([0.335859, -1.374087, -2.577824, -0.760478, 1.570796, 1.906656],accel_mss,speed_ms,0,blend_radius_m)
      movel([0.337030, -1.373968, -2.577907, -0.760514, 1.570796, 1.907827],accel_mss,speed_ms,0,blend_radius_m)
      movel([0.337336, -1.373947, -2.577922, -0.760521, 1.570796, 1.908132],accel_mss,speed_ms,0,blend_radius_m)
      movel([0.337636, -1.373942, -2.577925, -0.760522, 1.570796, 1.908432],accel_mss,speed_ms,0,blend_radius_m)
      movel([0.337928, -1.373953, -2.577917, -0.760519, 1.570796, 1.908724],accel_mss,speed_ms,0,blend_radius_m)
      movel([0.338213, -1.373981, -2.577898, -0.760510, 1.570796, 1.909010],accel_mss,speed_ms,0,blend_radius_m)
      movel([0.338485, -1.374028, -2.577865, -0.760496, 1.570796, 1.909281],accel_mss,speed_ms,0,blend_radius_m)
      speed_ms = 0.003
      movel([0.338485, -1.360932, -2.571804, -0.779653, 1.570796, 1.909281],accel_mss,speed_ms,0,blend_radius_m)
      speed_ms = 0.01
      movel([0.338485, -1.335837, -2.559287, -0.817264, 1.570796, 1.909281],accel_mss,speed_ms,0,blend_radius_m)
      movel([0.338648, -1.333404, -2.560884, -0.818101, 1.570796, 1.909444],accel_mss,speed_ms,0,blend_radius_m)
      movel([0.338648, -1.358541, -2.573431, -0.780417, 1.570796, 1.909444],accel_mss,speed_ms,0,blend_radius_m)
      speed_ms = 0.003
      movel([0.338648, -1.368346, -2.578002, -0.766041, 1.570796, 1.909444],accel_mss,speed_ms,0,blend_radius_m)
      speed_ms = 0.007
      movel([0.338233, -1.368407, -2.577960, -0.766022, 1.570796, 1.909029],accel_mss,speed_ms,0,blend_radius_m)
      movel([0.337823, -1.368456, -2.577926, -0.766007, 1.570796, 1.908619],accel_mss,speed_ms,0,blend_radius_m)
      movel([0.335051, -1.368741, -2.577729, -0.765918, 1.570796, 1.905847],accel_mss,speed_ms,0,blend_radius_m)
      movel([0.333043, -1.368967, -2.577574, -0.765849, 1.570796, 1.903840],accel_mss,speed_ms,0,blend_radius_m)
      movel([0.331056, -1.369230, -2.577392, -0.765767, 1.570796, 1.901852],accel_mss,speed_ms,0,blend_radius_m)
